DATA_BLOCK "1DB_simTT"   // DB999
{ S7_Optimized_Access := 'TRUE' }
VERSION : 0.1
   VAR
      TForSim : Array[0..359] of Int;   // Массив температур для эмуляции в формате Int
   END_VAR
BEGIN
   TForSim[0] := 200;
   TForSim[1] := 200;
   TForSim[2] := 199;
   TForSim[3] := 198;
   TForSim[4] := 197;
   TForSim[5] := 196;
   TForSim[6] := 196;
   TForSim[7] := 196;
   TForSim[8] := 196;
   TForSim[9] := 196;
   TForSim[10] := 195;
   TForSim[11] := 194;
   TForSim[12] := 194;
   TForSim[13] := 193;
   TForSim[14] := 193;
   TForSim[15] := 193;
   TForSim[16] := 193;
   TForSim[17] := 192;
   TForSim[18] := 192;
   TForSim[19] := 192;
   TForSim[20] := 192;
   TForSim[21] := 191;
   TForSim[22] := 191;
   TForSim[23] := 190;
   TForSim[24] := 189;
   TForSim[25] := 189;
   TForSim[26] := 189;
   TForSim[27] := 189;
   TForSim[28] := 188;
   TForSim[29] := 188;
   TForSim[30] := 187;
   TForSim[31] := 187;
   TForSim[32] := 187;
   TForSim[33] := 188;
   TForSim[34] := 188;
   TForSim[35] := 190;
   TForSim[36] := 190;
   TForSim[37] := 191;
   TForSim[38] := 191;
   TForSim[39] := 191;
   TForSim[40] := 193;
   TForSim[41] := 193;
   TForSim[42] := 193;
   TForSim[43] := 195;
   TForSim[44] := 195;
   TForSim[45] := 195;
   TForSim[46] := 196;
   TForSim[47] := 197;
   TForSim[48] := 198;
   TForSim[49] := 200;
   TForSim[50] := 200;
   TForSim[51] := 200;
   TForSim[52] := 201;
   TForSim[53] := 202;
   TForSim[54] := 203;
   TForSim[55] := 204;
   TForSim[56] := 205;
   TForSim[57] := 206;
   TForSim[58] := 207;
   TForSim[59] := 208;
   TForSim[60] := 209;
   TForSim[61] := 211;
   TForSim[62] := 211;
   TForSim[63] := 211;
   TForSim[64] := 211;
   TForSim[65] := 211;
   TForSim[66] := 210;
   TForSim[67] := 211;
   TForSim[68] := 211;
   TForSim[69] := 213;
   TForSim[70] := 214;
   TForSim[71] := 215;
   TForSim[72] := 215;
   TForSim[73] := 217;
   TForSim[74] := 218;
   TForSim[75] := 219;
   TForSim[76] := 220;
   TForSim[77] := 221;
   TForSim[78] := 222;
   TForSim[79] := 223;
   TForSim[80] := 225;
   TForSim[81] := 227;
   TForSim[82] := 230;
   TForSim[83] := 233;
   TForSim[84] := 236;
   TForSim[85] := 239;
   TForSim[86] := 241;
   TForSim[87] := 242;
   TForSim[88] := 244;
   TForSim[89] := 247;
   TForSim[90] := 249;
   TForSim[91] := 250;
   TForSim[92] := 250;
   TForSim[93] := 250;
   TForSim[94] := 250;
   TForSim[95] := 252;
   TForSim[96] := 254;
   TForSim[97] := 256;
   TForSim[98] := 257;
   TForSim[99] := 257;
   TForSim[100] := 259;
   TForSim[101] := 259;
   TForSim[102] := 259;
   TForSim[103] := 259;
   TForSim[104] := 260;
   TForSim[105] := 261;
   TForSim[106] := 261;
   TForSim[107] := 262;
   TForSim[108] := 262;
   TForSim[109] := 262;
   TForSim[110] := 263;
   TForSim[111] := 262;
   TForSim[112] := 262;
   TForSim[113] := 262;
   TForSim[114] := 262;
   TForSim[115] := 261;
   TForSim[116] := 261;
   TForSim[117] := 261;
   TForSim[118] := 261;
   TForSim[119] := 261;
   TForSim[120] := 260;
   TForSim[121] := 259;
   TForSim[122] := 259;
   TForSim[123] := 257;
   TForSim[124] := 256;
   TForSim[125] := 255;
   TForSim[126] := 254;
   TForSim[127] := 253;
   TForSim[128] := 253;
   TForSim[129] := 252;
   TForSim[130] := 252;
   TForSim[131] := 253;
   TForSim[132] := 253;
   TForSim[133] := 253;
   TForSim[134] := 252;
   TForSim[135] := 253;
   TForSim[136] := 253;
   TForSim[137] := 254;
   TForSim[138] := 255;
   TForSim[139] := 256;
   TForSim[140] := 259;
   TForSim[141] := 262;
   TForSim[142] := 264;
   TForSim[143] := 266;
   TForSim[144] := 266;
   TForSim[145] := 267;
   TForSim[146] := 267;
   TForSim[147] := 267;
   TForSim[148] := 270;
   TForSim[149] := 270;
   TForSim[150] := 271;
   TForSim[151] := 273;
   TForSim[152] := 273;
   TForSim[153] := 273;
   TForSim[154] := 274;
   TForSim[155] := 275;
   TForSim[156] := 275;
   TForSim[157] := 276;
   TForSim[158] := 277;
   TForSim[159] := 280;
   TForSim[160] := 281;
   TForSim[161] := 282;
   TForSim[162] := 282;
   TForSim[163] := 282;
   TForSim[164] := 284;
   TForSim[165] := 284;
   TForSim[166] := 285;
   TForSim[167] := 286;
   TForSim[168] := 286;
   TForSim[169] := 288;
   TForSim[170] := 288;
   TForSim[171] := 289;
   TForSim[172] := 291;
   TForSim[173] := 291;
   TForSim[174] := 292;
   TForSim[175] := 292;
   TForSim[176] := 292;
   TForSim[177] := 295;
   TForSim[178] := 294;
   TForSim[179] := 294;
   TForSim[180] := 295;
   TForSim[181] := 297;
   TForSim[182] := 298;
   TForSim[183] := 298;
   TForSim[184] := 300;
   TForSim[185] := 300;
   TForSim[186] := 300;
   TForSim[187] := 301;
   TForSim[188] := 301;
   TForSim[189] := 302;
   TForSim[190] := 303;
   TForSim[191] := 304;
   TForSim[192] := 304;
   TForSim[193] := 304;
   TForSim[194] := 306;
   TForSim[195] := 306;
   TForSim[196] := 306;
   TForSim[197] := 308;
   TForSim[198] := 307;
   TForSim[199] := 307;
   TForSim[200] := 309;
   TForSim[201] := 310;
   TForSim[202] := 311;
   TForSim[203] := 311;
   TForSim[204] := 312;
   TForSim[205] := 312;
   TForSim[206] := 312;
   TForSim[207] := 314;
   TForSim[208] := 313;
   TForSim[209] := 314;
   TForSim[210] := 314;
   TForSim[211] := 315;
   TForSim[212] := 315;
   TForSim[213] := 312;
   TForSim[214] := 312;
   TForSim[215] := 312;
   TForSim[216] := 312;
   TForSim[217] := 315;
   TForSim[218] := 315;
   TForSim[219] := 314;
   TForSim[220] := 313;
   TForSim[221] := 312;
   TForSim[222] := 311;
   TForSim[223] := 311;
   TForSim[224] := 311;
   TForSim[225] := 311;
   TForSim[226] := 311;
   TForSim[227] := 308;
   TForSim[228] := 309;
   TForSim[229] := 309;
   TForSim[230] := 308;
   TForSim[231] := 306;
   TForSim[232] := 305;
   TForSim[233] := 305;
   TForSim[234] := 303;
   TForSim[235] := 302;
   TForSim[236] := 302;
   TForSim[237] := 302;
   TForSim[238] := 301;
   TForSim[239] := 301;
   TForSim[240] := 301;
   TForSim[241] := 300;
   TForSim[242] := 299;
   TForSim[243] := 298;
   TForSim[244] := 297;
   TForSim[245] := 297;
   TForSim[246] := 297;
   TForSim[247] := 295;
   TForSim[248] := 295;
   TForSim[249] := 293;
   TForSim[250] := 293;
   TForSim[251] := 293;
   TForSim[252] := 290;
   TForSim[253] := 290;
   TForSim[254] := 289;
   TForSim[255] := 289;
   TForSim[256] := 289;
   TForSim[257] := 289;
   TForSim[258] := 290;
   TForSim[259] := 291;
   TForSim[260] := 292;
   TForSim[261] := 293;
   TForSim[262] := 294;
   TForSim[263] := 294;
   TForSim[264] := 295;
   TForSim[265] := 297;
   TForSim[266] := 298;
   TForSim[267] := 300;
   TForSim[268] := 301;
   TForSim[269] := 301;
   TForSim[270] := 302;
   TForSim[271] := 304;
   TForSim[272] := 304;
   TForSim[273] := 303;
   TForSim[274] := 301;
   TForSim[275] := 298;
   TForSim[276] := 299;
   TForSim[277] := 298;
   TForSim[278] := 296;
   TForSim[279] := 295;
   TForSim[280] := 295;
   TForSim[281] := 295;
   TForSim[282] := 294;
   TForSim[283] := 293;
   TForSim[284] := 292;
   TForSim[285] := 292;
   TForSim[286] := 290;
   TForSim[287] := 290;
   TForSim[288] := 287;
   TForSim[289] := 288;
   TForSim[290] := 288;
   TForSim[291] := 288;
   TForSim[292] := 286;
   TForSim[293] := 286;
   TForSim[294] := 284;
   TForSim[295] := 283;
   TForSim[296] := 280;
   TForSim[297] := 280;
   TForSim[298] := 278;
   TForSim[299] := 277;
   TForSim[300] := 276;
   TForSim[301] := 275;
   TForSim[302] := 274;
   TForSim[303] := 271;
   TForSim[304] := 272;
   TForSim[305] := 272;
   TForSim[306] := 270;
   TForSim[307] := 267;
   TForSim[308] := 265;
   TForSim[309] := 263;
   TForSim[310] := 261;
   TForSim[311] := 260;
   TForSim[312] := 258;
   TForSim[313] := 256;
   TForSim[314] := 254;
   TForSim[315] := 251;
   TForSim[316] := 252;
   TForSim[317] := 252;
   TForSim[318] := 253;
   TForSim[319] := 253;
   TForSim[320] := 251;
   TForSim[321] := 251;
   TForSim[322] := 249;
   TForSim[323] := 247;
   TForSim[324] := 246;
   TForSim[325] := 244;
   TForSim[326] := 242;
   TForSim[327] := 240;
   TForSim[328] := 238;
   TForSim[329] := 236;
   TForSim[330] := 233;
   TForSim[331] := 231;
   TForSim[332] := 229;
   TForSim[333] := 227;
   TForSim[334] := 225;
   TForSim[335] := 223;
   TForSim[336] := 222;
   TForSim[337] := 220;
   TForSim[338] := 219;
   TForSim[339] := 218;
   TForSim[340] := 217;
   TForSim[341] := 217;
   TForSim[342] := 217;
   TForSim[343] := 216;
   TForSim[344] := 215;
   TForSim[345] := 214;
   TForSim[346] := 214;
   TForSim[347] := 214;
   TForSim[348] := 213;
   TForSim[349] := 212;
   TForSim[350] := 210;
   TForSim[351] := 208;
   TForSim[352] := 206;
   TForSim[353] := 204;
   TForSim[354] := 203;
   TForSim[355] := 203;
   TForSim[356] := 203;
   TForSim[357] := 202;
   TForSim[358] := 202;
   TForSim[359] := 200;
END_DATA_BLOCK

// folder: System blocks/Program resources

DATA_BLOCK "Timer_2_DB"   // DB2
{ S7_Optimized_Access := 'TRUE' }
AUTHOR : Simatic
FAMILY : IEC
NAME : IEC_TMR
VERSION : 1.0
// stored: InstanceOfName IEC_TIMER
"IEC_TIMER"
BEGIN
END_DATA_BLOCK

DATA_BLOCK "IEC_Timer_1"   // DB601
{ S7_Optimized_Access := 'TRUE' }
AUTHOR : Simatic
FAMILY : IEC
NAME : IEC_TMR
VERSION : 1.0
// stored: InstanceOfName IEC_TIMER
"IEC_TIMER"
BEGIN
END_DATA_BLOCK

DATA_BLOCK "IEC_Timer_2"   // DB602
{ S7_Optimized_Access := 'TRUE' }
AUTHOR : Simatic
FAMILY : IEC
NAME : IEC_TMR
VERSION : 1.0
// stored: InstanceOfName IEC_TIMER
"IEC_TIMER"
BEGIN
END_DATA_BLOCK

DATA_BLOCK "IEC_Timer_3"   // DB603
{ S7_Optimized_Access := 'TRUE' }
AUTHOR : Simatic
FAMILY : IEC
NAME : IEC_TMR
VERSION : 1.0
// stored: InstanceOfName IEC_TIMER
"IEC_TIMER"
BEGIN
END_DATA_BLOCK

DATA_BLOCK "IEC_Timer_4"   // DB604
{ S7_Optimized_Access := 'TRUE' }
AUTHOR : Simatic
FAMILY : IEC
NAME : IEC_TMR
VERSION : 1.0
// stored: InstanceOfName IEC_TIMER
"IEC_TIMER"
BEGIN
END_DATA_BLOCK

DATA_BLOCK "IEC_Timer_5"   // DB605
{ S7_Optimized_Access := 'TRUE' }
AUTHOR : Simatic
FAMILY : IEC
NAME : IEC_TMR
VERSION : 1.0
// stored: InstanceOfName IEC_TIMER
"IEC_TIMER"
BEGIN
END_DATA_BLOCK

DATA_BLOCK "IEC_Timer_6"   // DB606
{ S7_Optimized_Access := 'TRUE' }
AUTHOR : Simatic
FAMILY : IEC
NAME : IEC_TMR
VERSION : 1.0
// stored: InstanceOfName IEC_TIMER
"IEC_TIMER"
BEGIN
END_DATA_BLOCK

DATA_BLOCK "IEC_Timer_7"   // DB607
{ S7_Optimized_Access := 'TRUE' }
AUTHOR : Simatic
FAMILY : IEC
NAME : IEC_TMR
VERSION : 1.0
// stored: InstanceOfName IEC_TIMER
"IEC_TIMER"
BEGIN
END_DATA_BLOCK

DATA_BLOCK "IEC_Timer_8"   // DB608
{ S7_Optimized_Access := 'TRUE' }
AUTHOR : Simatic
FAMILY : IEC
NAME : IEC_TMR
VERSION : 1.0
// stored: InstanceOfName IEC_TIMER
"IEC_TIMER"
BEGIN
END_DATA_BLOCK

DATA_BLOCK "SimTimer11"   // DB911
{ S7_Optimized_Access := 'TRUE' }
AUTHOR : Simatic
FAMILY : IEC
NAME : IEC_TMR
VERSION : 1.0
// stored: InstanceOfName IEC_TIMER
"IEC_TIMER"
BEGIN
END_DATA_BLOCK

DATA_BLOCK "SimTimer12"   // DB912
{ S7_Optimized_Access := 'TRUE' }
AUTHOR : Simatic
FAMILY : IEC
NAME : IEC_TMR
VERSION : 1.0
// stored: InstanceOfName IEC_TIMER
"IEC_TIMER"
BEGIN
END_DATA_BLOCK

DATA_BLOCK "SimTimer21"   // DB921
{ S7_Optimized_Access := 'TRUE' }
AUTHOR : Simatic
FAMILY : IEC
NAME : IEC_TMR
VERSION : 1.0
// stored: InstanceOfName IEC_TIMER
"IEC_TIMER"
BEGIN
END_DATA_BLOCK

DATA_BLOCK "SimTimer22"   // DB922
{ S7_Optimized_Access := 'TRUE' }
AUTHOR : Simatic
FAMILY : IEC
NAME : IEC_TMR
VERSION : 1.0
// stored: InstanceOfName IEC_TIMER
"IEC_TIMER"
BEGIN
END_DATA_BLOCK

// folder: (top level)

ORGANIZATION_BLOCK "1Main"   // OB1, LAD, ProgramCycle
TITLE = "Main Program Sweep (Cycle)"
{ S7_Optimized_Access := 'TRUE' }
VERSION : 0.1
// ОВ1 - главная циклическая программа. Вызывается операционной системой CPU
   VAR_INPUT
      Initial_Call : Bool;   // Initial call of this OB
      Remanence : Bool;   // =True, if remanent data are available
   END_VAR
   VAR_TEMP
      txExtStopVE : Bool;   // Внешняя блокировка дымососа по вибрации
      txExtStopTEB : Bool;   // Внешняя блокировка дымососа по т-ре подшипников
      txExtStopTEW : Bool;   // Внешняя блокировка дымососа по т-ре обмоток
      trValue : Real;   // Временная переменная типа Real
   END_VAR
BEGIN

REGION Network 2: Зеркалирование дискретных входов
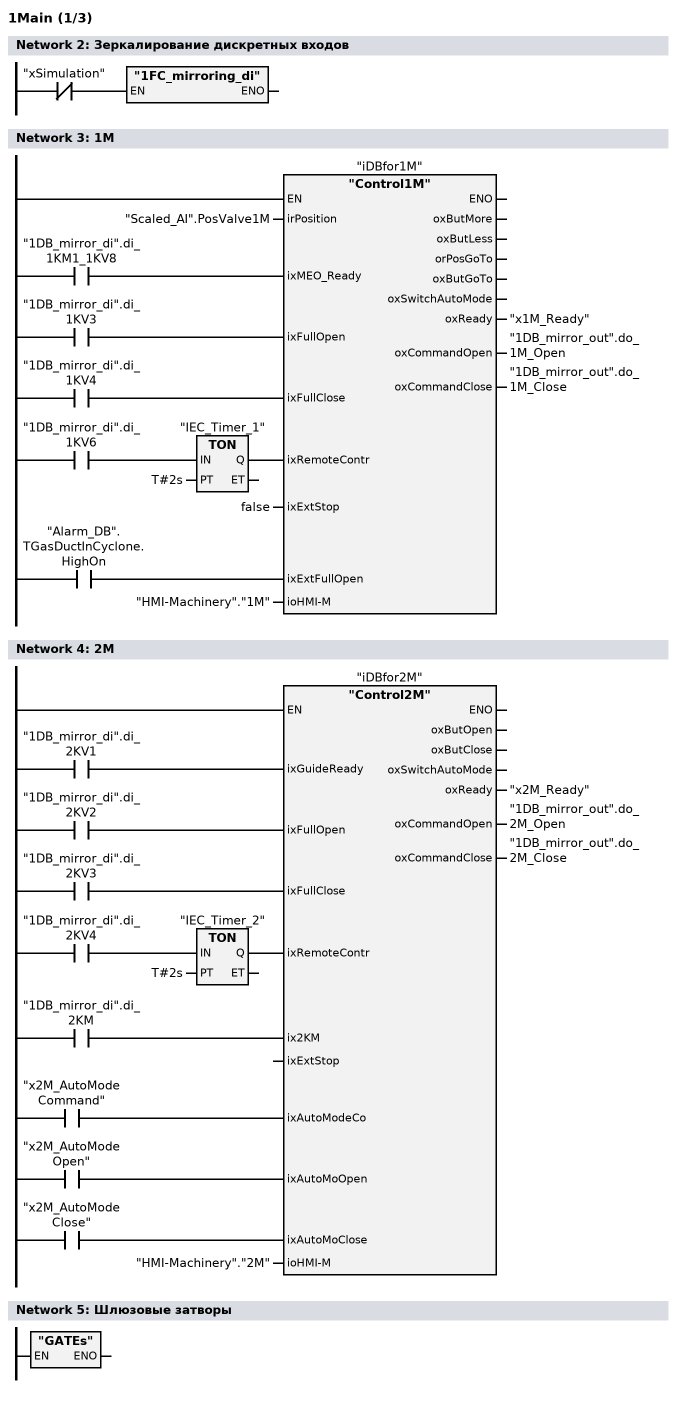
   RUNG wire#powerrail
      I_Contact( "xSimulation" )
      "1FC_mirroring_di"()
   END_RUNG
   // the same network as SCL:
   IF NOT "xSimulation" THEN "1FC_mirroring_di"(); END_IF;
END_REGION

REGION Network 3: 1M
   "IEC_Timer_1".TON(IN := "1DB_mirror_di".di_1KV6, PT := T#2s);
   "iDBfor1M"(irPosition := "Scaled_AI".PosValve1M,   // "Control1M"
              ixMEO_Ready := "1DB_mirror_di".di_1KM1_1KV8,
              ixFullOpen := "1DB_mirror_di".di_1KV3,
              ixFullClose := "1DB_mirror_di".di_1KV4,
              ixRemoteContr := "IEC_Timer_1".Q,
              ixExtStop := false,
              ixExtFullOpen := "Alarm_DB".TGasDuctInCyclone.HighOn,
              "ioHMI-M" := "HMI-Machinery"."1M",
              oxReady => "x1M_Ready",
              oxCommandOpen => "1DB_mirror_out".do_1M_Open,
              oxCommandClose => "1DB_mirror_out".do_1M_Close);
END_REGION

REGION Network 4: 2M
   "IEC_Timer_2".TON(IN := "1DB_mirror_di".di_2KV4, PT := T#2s);
   "iDBfor2M"(ixGuideReady := "1DB_mirror_di".di_2KV1,   // "Control2M"
              ixFullOpen := "1DB_mirror_di".di_2KV2,
              ixFullClose := "1DB_mirror_di".di_2KV3,
              ixRemoteContr := "IEC_Timer_2".Q,
              ix2KM := "1DB_mirror_di".di_2KM,
              ixAutoModeCo := "x2M_AutoModeCommand",
              ixAutoMoOpen := "x2M_AutoModeOpen",
              ixAutoMoClose := "x2M_AutoModeClose",
              "ioHMI-M" := "HMI-Machinery"."2M",
              oxReady => "x2M_Ready",
              oxCommandOpen => "1DB_mirror_out".do_2M_Open,
              oxCommandClose => "1DB_mirror_out".do_2M_Close);
END_REGION

REGION Network 5: Шлюзовые затворы
   RUNG wire#powerrail
      "GATEs"()
   END_RUNG
   // the same network as SCL:
   "GATEs"();
END_REGION

REGION Network 7: Подготовка внешних блокировок дымососа (14 шт.)
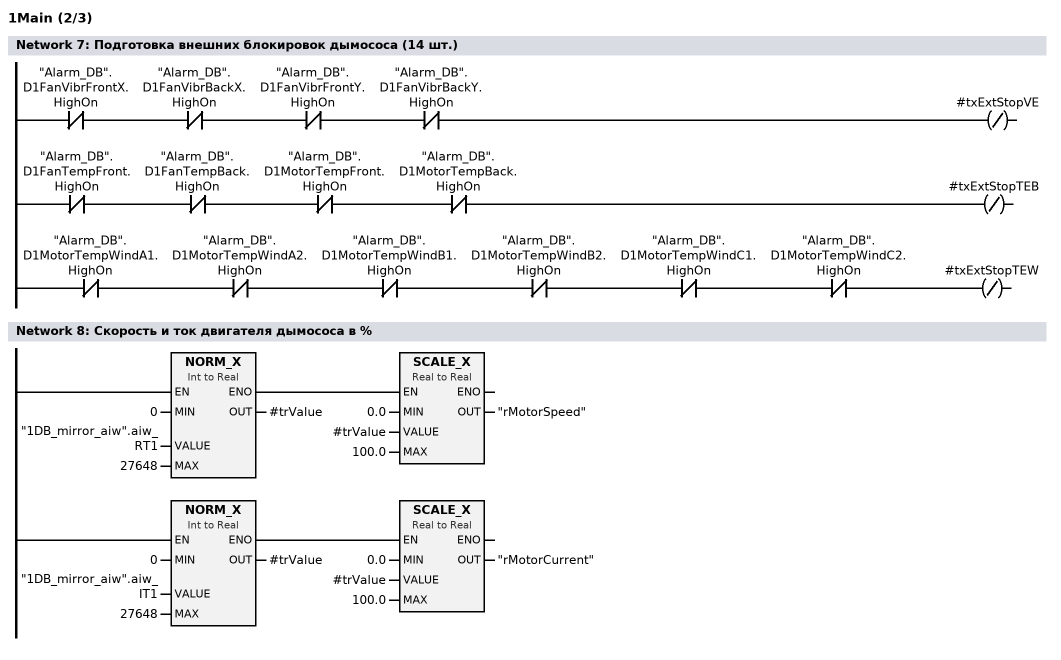
   RUNG wire#powerrail
      I_Contact( "Alarm_DB".D1FanVibrFrontX.HighOn )
      I_Contact( "Alarm_DB".D1FanVibrBackX.HighOn )
      I_Contact( "Alarm_DB".D1FanVibrFrontY.HighOn )
      I_Contact( "Alarm_DB".D1FanVibrBackY.HighOn )
      I_Coil( #txExtStopVE )
   END_RUNG
   RUNG wire#powerrail
      I_Contact( "Alarm_DB".D1FanTempFront.HighOn )
      I_Contact( "Alarm_DB".D1FanTempBack.HighOn )
      I_Contact( "Alarm_DB".D1MotorTempFront.HighOn )
      I_Contact( "Alarm_DB".D1MotorTempBack.HighOn )
      I_Coil( #txExtStopTEB )
   END_RUNG
   RUNG wire#powerrail
      I_Contact( "Alarm_DB".D1MotorTempWindA1.HighOn )
      I_Contact( "Alarm_DB".D1MotorTempWindA2.HighOn )
      I_Contact( "Alarm_DB".D1MotorTempWindB1.HighOn )
      I_Contact( "Alarm_DB".D1MotorTempWindB2.HighOn )
      I_Contact( "Alarm_DB".D1MotorTempWindC1.HighOn )
      I_Contact( "Alarm_DB".D1MotorTempWindC2.HighOn )
      I_Coil( #txExtStopTEW )
   END_RUNG
   // the same network as SCL:
   #txExtStopVE := NOT (NOT "Alarm_DB".D1FanVibrFrontX.HighOn AND NOT "Alarm_DB".D1FanVibrBackX.HighOn AND NOT "Alarm_DB".D1FanVibrFrontY.HighOn AND NOT "Alarm_DB".D1FanVibrBackY.HighOn);
   #txExtStopTEB := NOT (NOT "Alarm_DB".D1FanTempFront.HighOn AND NOT "Alarm_DB".D1FanTempBack.HighOn AND NOT "Alarm_DB".D1MotorTempFront.HighOn AND NOT "Alarm_DB".D1MotorTempBack.HighOn);
   #txExtStopTEW := NOT (NOT "Alarm_DB".D1MotorTempWindA1.HighOn AND NOT "Alarm_DB".D1MotorTempWindA2.HighOn AND NOT "Alarm_DB".D1MotorTempWindB1.HighOn AND NOT "Alarm_DB".D1MotorTempWindB2.HighOn AND NOT "Alarm_DB".D1MotorTempWindC1.HighOn AND NOT "Alarm_DB".D1MotorTempWindC2.HighOn);
END_REGION

REGION Network 8: Скорость и ток двигателя дымососа в %
   RUNG wire#powerrail
      { S7_Templates := "[SrcType := Int, DestType := Real]" } Normalize(min := 0, value := "1DB_mirror_aiw".aiw_RT1, max := 27648, out => #trValue)
      { S7_Templates := "[SrcType := Real, DestType := Real]" } Scale(min := 0.0, value := #trValue, max := 100.0, out => "rMotorSpeed")
   END_RUNG
   RUNG wire#powerrail
      { S7_Templates := "[SrcType := Int, DestType := Real]" } Normalize(min := 0, value := "1DB_mirror_aiw".aiw_IT1, max := 27648, out => #trValue)
      { S7_Templates := "[SrcType := Real, DestType := Real]" } Scale(min := 0.0, value := #trValue, max := 100.0, out => "rMotorCurrent")
   END_RUNG
   // the same network as SCL:
   #trValue := NORM_X(MIN := 0, VALUE := "1DB_mirror_aiw".aiw_RT1, MAX := 27648);
   "rMotorSpeed" := SCALE_X(MIN := 0.0, VALUE := #trValue, MAX := 100.0);
   #trValue := NORM_X(MIN := 0, VALUE := "1DB_mirror_aiw".aiw_IT1, MAX := 27648);
   "rMotorCurrent" := SCALE_X(MIN := 0.0, VALUE := #trValue, MAX := 100.0);
END_REGION

REGION Network 9: Дымосос
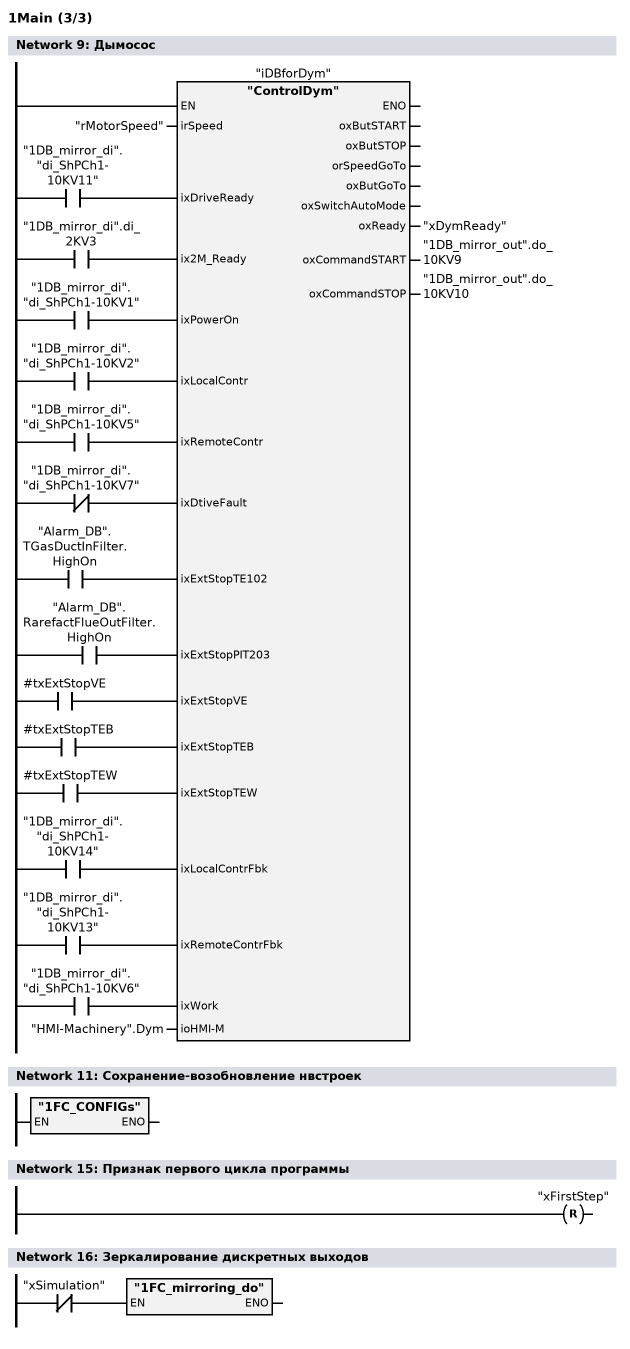
   RUNG wire#powerrail
      "iDBforDym"(ixDriveReady := wire#w1, ix2M_Ready := wire#w2, ixPowerOn := wire#w3, ixLocalContr := wire#w4, ixRemoteContr := wire#w5, ixDtiveFault := wire#w6, ixExtStopTE102 := wire#w7, ixExtStopРІТ203 := wire#w8, ixExtStopVE := wire#w9, ixExtStopTEB := wire#w10, ixExtStopTEW := wire#w11, ixLocalContrFbk := wire#w12, ixRemoteContrFbk := wire#w13, ixWork := wire#w14, irSpeed := "rMotorSpeed", "ioHMI-M" := "HMI-Machinery".Dym, oxButSTART =>, oxButSTOP =>, orSpeedGoTo =>, oxButGoTo =>, oxSwitchAutoMode =>, oxReady => "xDymReady", oxCommandSTART => "1DB_mirror_out".do_10KV9, oxCommandSTOP => "1DB_mirror_out".do_10KV10)
   END_RUNG
   RUNG wire#powerrail
      Contact( "1DB_mirror_di"."di_ShPCh1-10KV11" )
   END_RUNG wire#w1
   RUNG wire#powerrail
      Contact( "1DB_mirror_di".di_2KV3 )
   END_RUNG wire#w2
   RUNG wire#powerrail
      Contact( "1DB_mirror_di"."di_ShPCh1-10KV1" )
   END_RUNG wire#w3
   RUNG wire#powerrail
      Contact( "1DB_mirror_di"."di_ShPCh1-10KV2" )
   END_RUNG wire#w4
   RUNG wire#powerrail
      Contact( "1DB_mirror_di"."di_ShPCh1-10KV5" )
   END_RUNG wire#w5
   RUNG wire#powerrail
      I_Contact( "1DB_mirror_di"."di_ShPCh1-10KV7" )
   END_RUNG wire#w6
   RUNG wire#powerrail
      Contact( "Alarm_DB".TGasDuctInFilter.HighOn )
   END_RUNG wire#w7
   RUNG wire#powerrail
      Contact( "Alarm_DB".RarefactFlueOutFilter.HighOn )
   END_RUNG wire#w8
   RUNG wire#powerrail
      Contact( #txExtStopVE )
   END_RUNG wire#w9
   RUNG wire#powerrail
      Contact( #txExtStopTEB )
   END_RUNG wire#w10
   RUNG wire#powerrail
      Contact( #txExtStopTEW )
   END_RUNG wire#w11
   RUNG wire#powerrail
      Contact( "1DB_mirror_di"."di_ShPCh1-10KV14" )
   END_RUNG wire#w12
   RUNG wire#powerrail
      Contact( "1DB_mirror_di"."di_ShPCh1-10KV13" )
   END_RUNG wire#w13
   RUNG wire#powerrail
      Contact( "1DB_mirror_di"."di_ShPCh1-10KV6" )
   END_RUNG wire#w14
   // the same network as SCL:
   "iDBforDym"(irSpeed := "rMotorSpeed",   // "ControlDym"
               ixDriveReady := "1DB_mirror_di"."di_ShPCh1-10KV11",
               ix2M_Ready := "1DB_mirror_di".di_2KV3,
               ixPowerOn := "1DB_mirror_di"."di_ShPCh1-10KV1",
               ixLocalContr := "1DB_mirror_di"."di_ShPCh1-10KV2",
               ixRemoteContr := "1DB_mirror_di"."di_ShPCh1-10KV5",
               ixDtiveFault := NOT "1DB_mirror_di"."di_ShPCh1-10KV7",
               ixExtStopTE102 := "Alarm_DB".TGasDuctInFilter.HighOn,
               ixExtStopРІТ203 := "Alarm_DB".RarefactFlueOutFilter.HighOn,
               ixExtStopVE := #txExtStopVE,
               ixExtStopTEB := #txExtStopTEB,
               ixExtStopTEW := #txExtStopTEW,
               ixLocalContrFbk := "1DB_mirror_di"."di_ShPCh1-10KV14",
               ixRemoteContrFbk := "1DB_mirror_di"."di_ShPCh1-10KV13",
               ixWork := "1DB_mirror_di"."di_ShPCh1-10KV6",
               "ioHMI-M" := "HMI-Machinery".Dym,
               oxReady => "xDymReady",
               oxCommandSTART => "1DB_mirror_out".do_10KV9,
               oxCommandSTOP => "1DB_mirror_out".do_10KV10);
END_REGION

REGION Network 11: Сохранение-возобновление нвстроек
   RUNG wire#powerrail
      "1FC_CONFIGs"()
   END_RUNG
   // the same network as SCL:
   "1FC_CONFIGs"();
END_REGION

REGION Network 14: Все NW что ниже должны быть в конце ОВ1:
END_REGION

REGION Network 15: Признак первого цикла программы
   RUNG wire#powerrail
      R_Coil( "xFirstStep" )
   END_RUNG
   // the same network as SCL:
   "xFirstStep" := FALSE;
END_REGION

REGION Network 16: Зеркалирование дискретных выходов
   RUNG wire#powerrail
      I_Contact( "xSimulation" )
      "1FC_mirroring_do"()
   END_RUNG
   // the same network as SCL:
   IF NOT "xSimulation" THEN "1FC_mirroring_do"(); END_IF;
END_REGION
END_ORGANIZATION_BLOCK

ORGANIZATION_BLOCK "1Cyclic irupt_100"   // OB30, LAD, CyclicInterrupt
TITLE = "Cyclic interrupt"
{ S7_Optimized_Access := 'TRUE' }
VERSION : 0.1
// ОВ30 настроен на циклический вызов каждые 100 милисекунд. 
// Вызывается операционной системой CPU
   VAR_INPUT
      Initial_Call : Bool;   // Initial call of this OB
      Event_Count : Int;   // Events discarded
   END_VAR
   VAR_TEMP
      trForRegeneration : Real;   // Разность разрежений
      tiDymPID_Command : Int;   // Для задания скорости приводу дымососа от ПИДа
   END_VAR
   VAR_TEMP   // added for the SCL form of the ladder/FBD networks
      _w1 : Bool;
      _w2 : Bool;
      _w3 : Bool;
      _w4 : Bool;
   END_VAR
BEGIN

REGION Network 2: Симуляция механизмов
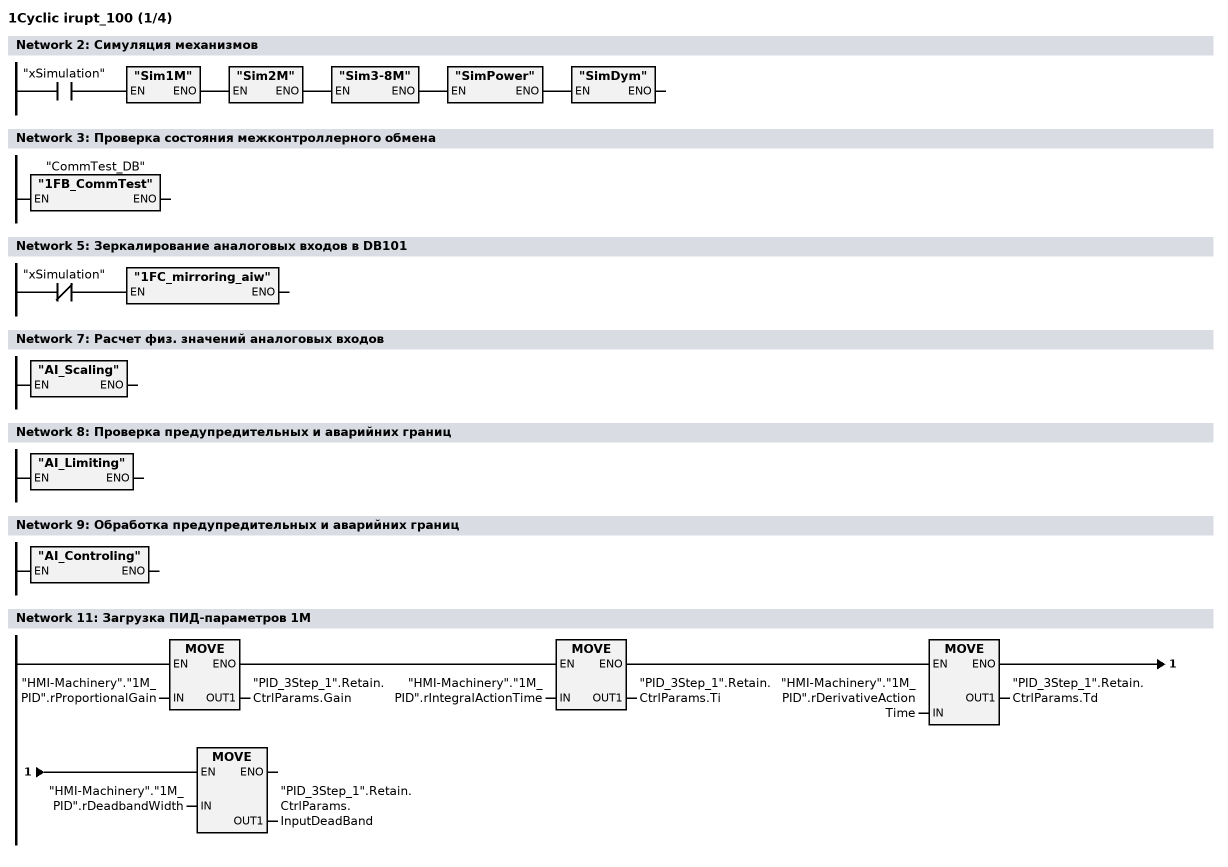
   RUNG wire#powerrail
      Contact( "xSimulation" )
      "Sim1M"()
      "Sim2M"()
      "Sim3-8M"()
      "SimPower"()
      "SimDym"()
   END_RUNG
   // the same network as SCL:
   "Sim1M"(EN := "xSimulation", ENO => #_w1);
   "Sim2M"(EN := #_w1, ENO => #_w2);
   "Sim3-8M"(EN := #_w2, ENO => #_w3);
   "SimPower"(EN := #_w3, ENO => #_w4);
   IF #_w4 THEN "SimDym"(); END_IF;
END_REGION

REGION Network 3: Проверка состояния межконтроллерного обмена
   RUNG wire#powerrail
      "CommTest_DB"()
   END_RUNG
   // the same network as SCL:
   "CommTest_DB"();   // "1FB_CommTest"
END_REGION

REGION Network 5: Зеркалирование аналоговых входов в DB101
   RUNG wire#powerrail
      I_Contact( "xSimulation" )
      "1FC_mirroring_aiw"()
   END_RUNG
   // the same network as SCL:
   IF NOT "xSimulation" THEN "1FC_mirroring_aiw"(); END_IF;
END_REGION

REGION Network 6: Обработка аналоговых входов (networks 4-6)
END_REGION

REGION Network 7: Расчет физ. значений аналоговых входов
   RUNG wire#powerrail
      "AI_Scaling"()
   END_RUNG
   // the same network as SCL:
   "AI_Scaling"();
END_REGION

REGION Network 8: Проверка предупредительных и аварийних границ
   RUNG wire#powerrail
      "AI_Limiting"()
   END_RUNG
   // the same network as SCL:
   "AI_Limiting"();
END_REGION

REGION Network 9: Обработка предупредительных и аварийних границ
   RUNG wire#powerrail
      "AI_Controling"()
   END_RUNG
   // the same network as SCL:
   "AI_Controling"();
END_REGION

REGION Network 11: Загрузка ПИД-параметров 1M
   RUNG wire#powerrail
      Move(in := "HMI-Machinery"."1M_PID".rProportionalGain, out1 => "PID_3Step_1".Retain.CtrlParams.Gain)
      Move(in := "HMI-Machinery"."1M_PID".rIntegralActionTime, out1 => "PID_3Step_1".Retain.CtrlParams.Ti)
      Move(in := "HMI-Machinery"."1M_PID".rDerivativeActionTime, out1 => "PID_3Step_1".Retain.CtrlParams.Td)
      Move(in := "HMI-Machinery"."1M_PID".rDeadbandWidth, out1 => "PID_3Step_1".Retain.CtrlParams.InputDeadBand)
   END_RUNG
   // the same network as SCL:
   "PID_3Step_1".Retain.CtrlParams.Gain := "HMI-Machinery"."1M_PID".rProportionalGain;
   "PID_3Step_1".Retain.CtrlParams.Ti := "HMI-Machinery"."1M_PID".rIntegralActionTime;
   "PID_3Step_1".Retain.CtrlParams.Td := "HMI-Machinery"."1M_PID".rDerivativeActionTime;
   "PID_3Step_1".Retain.CtrlParams.InputDeadBand := "HMI-Machinery"."1M_PID".rDeadbandWidth;
END_REGION

REGION Network 12: ПИД-регурятор для 1М
   // Жоден з цих трьох ПІДів (що нижче) не працюють у PLCSIM. Одже остаточне налагодження можливе тільке на майданчику
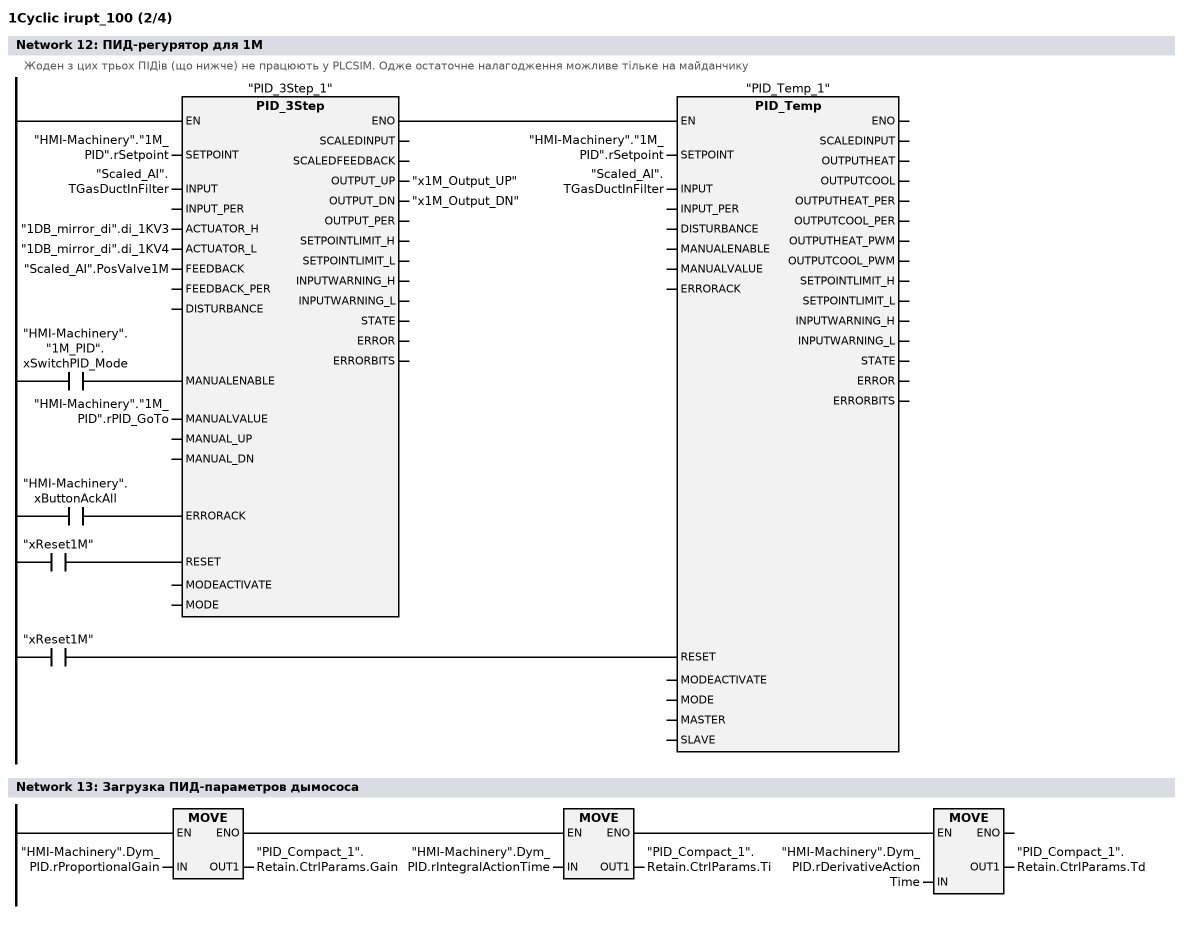
   // ENO of a box is taken as its EN; it also drops when the box reports an error
   "PID_3Step_1"(Setpoint := "HMI-Machinery"."1M_PID".rSetpoint,   // PID_3Step
                 Input := "Scaled_AI".TGasDuctInFilter,
                 Actuator_H := "1DB_mirror_di".di_1KV3,
                 Actuator_L := "1DB_mirror_di".di_1KV4,
                 Feedback := "Scaled_AI".PosValve1M,
                 ManualEnable := "HMI-Machinery"."1M_PID".xSwitchPID_Mode,
                 ManualValue := "HMI-Machinery"."1M_PID".rPID_GoTo,
                 ErrorAck := "HMI-Machinery".xButtonAckAll,
                 Reset := "xReset1M",
                 Output_UP => "x1M_Output_UP",
                 Output_DN => "x1M_Output_DN");
   "PID_Temp_1"(Setpoint := "HMI-Machinery"."1M_PID".rSetpoint,   // PID_Temp
                Input := "Scaled_AI".TGasDuctInFilter,
                Reset := "xReset1M");
END_REGION

REGION Network 13: Загрузка ПИД-параметров дымососа
   RUNG wire#powerrail
      Move(in := "HMI-Machinery".Dym_PID.rProportionalGain, out1 => "PID_Compact_1".Retain.CtrlParams.Gain)
      Move(in := "HMI-Machinery".Dym_PID.rIntegralActionTime, out1 => "PID_Compact_1".Retain.CtrlParams.Ti)
      Move(in := "HMI-Machinery".Dym_PID.rDerivativeActionTime, out1 => "PID_Compact_1".Retain.CtrlParams.Td)
   END_RUNG
   // the same network as SCL:
   "PID_Compact_1".Retain.CtrlParams.Gain := "HMI-Machinery".Dym_PID.rProportionalGain;
   "PID_Compact_1".Retain.CtrlParams.Ti := "HMI-Machinery".Dym_PID.rIntegralActionTime;
   "PID_Compact_1".Retain.CtrlParams.Td := "HMI-Machinery".Dym_PID.rDerivativeActionTime;
END_REGION

REGION Network 14: ПИД-регурятор для дымососа
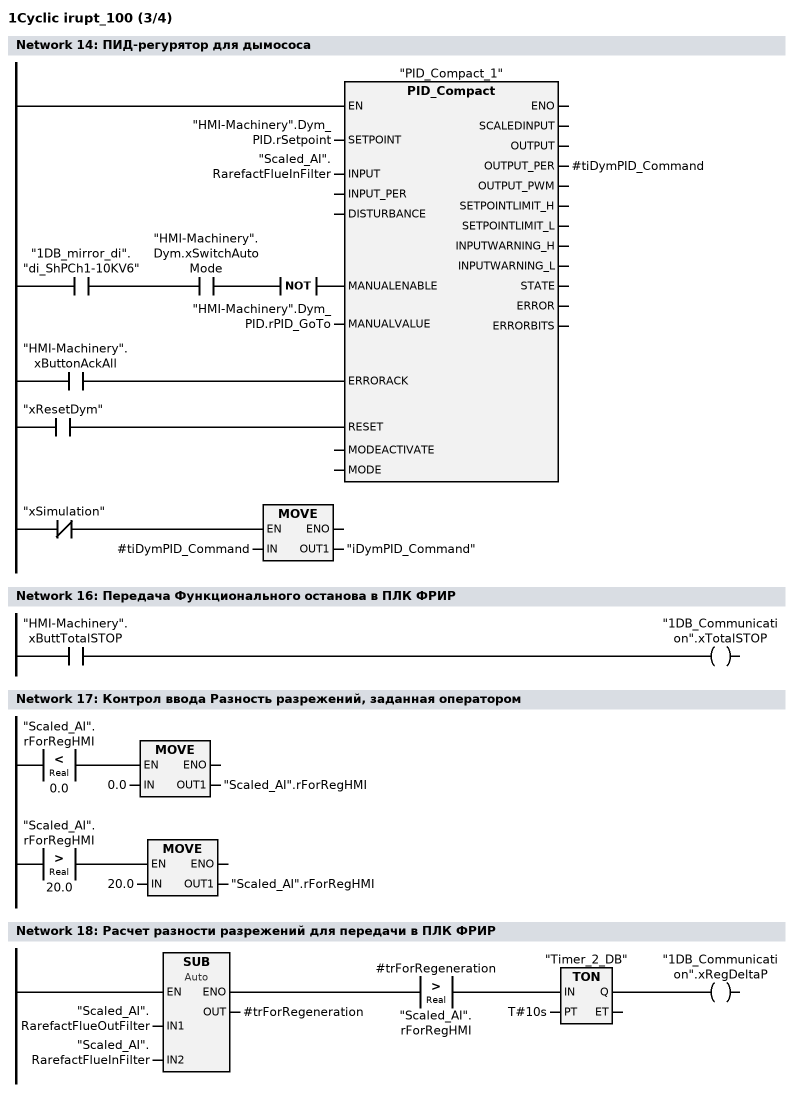
   "PID_Compact_1"(Setpoint := "HMI-Machinery".Dym_PID.rSetpoint,   // PID_Compact
                   Input := "Scaled_AI".RarefactFlueInFilter,
                   ManualEnable := NOT ("1DB_mirror_di"."di_ShPCh1-10KV6" AND "HMI-Machinery".Dym.xSwitchAutoMode),
                   ManualValue := "HMI-Machinery".Dym_PID.rPID_GoTo,
                   ErrorAck := "HMI-Machinery".xButtonAckAll,
                   Reset := "xResetDym",
                   Output_PER => #tiDymPID_Command);
   IF NOT "xSimulation" THEN "iDymPID_Command" := #tiDymPID_Command; END_IF;
END_REGION

REGION Network 16: Передача Функционального останова в ПЛК ФРИР
   RUNG wire#powerrail
      Contact( "HMI-Machinery".xButtTotalSTOP )
      Coil( "1DB_Communication".xTotalSTOP )
   END_RUNG
   // the same network as SCL:
   "1DB_Communication".xTotalSTOP := "HMI-Machinery".xButtTotalSTOP;
END_REGION

REGION Network 17: Контрол ввода Разность разрежений, заданная оператором
   RUNG wire#powerrail
      { S7_Templates := "SrcType := Real" } LT_Contact(in1 := "Scaled_AI".rForRegHMI, in2 := 0.0)
      Move(in := 0.0, out1 => "Scaled_AI".rForRegHMI)
   END_RUNG
   RUNG wire#powerrail
      { S7_Templates := "SrcType := Real" } GT_Contact(in1 := "Scaled_AI".rForRegHMI, in2 := 20.0)
      Move(in := 20.0, out1 => "Scaled_AI".rForRegHMI)
   END_RUNG
   // the same network as SCL:
   IF "Scaled_AI".rForRegHMI < 0.0 THEN "Scaled_AI".rForRegHMI := 0.0; END_IF;
   IF "Scaled_AI".rForRegHMI > 20.0 THEN "Scaled_AI".rForRegHMI := 20.0; END_IF;
END_REGION

REGION Network 18: Расчет разности разрежений для передачи в ПЛК ФРИР
   #trForRegeneration := "Scaled_AI".RarefactFlueOutFilter - "Scaled_AI".RarefactFlueInFilter;
   "Timer_2_DB".TON(IN := #trForRegeneration > "Scaled_AI".rForRegHMI, PT := T#10s);
   "1DB_Communication".xRegDeltaP := "Timer_2_DB".Q;
END_REGION

REGION Network 19: Передача данных в контроллер ФРИР
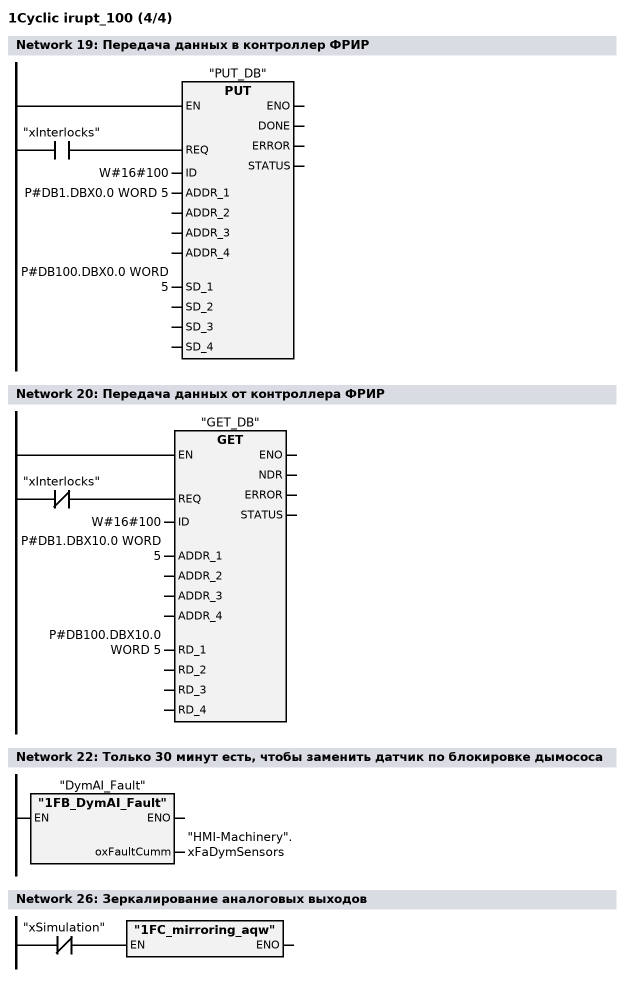
   "PUT_DB"(REQ := "xInterlocks", ID := W#16#100, ADDR_1 := P#DB1.DBX0.0 WORD 5, SD_1 := P#DB100.DBX0.0 WORD 5);   // PUT
END_REGION

REGION Network 20: Передача данных от контроллера ФРИР
   "GET_DB"(REQ := NOT "xInterlocks",   // GET
            ID := W#16#100,
            ADDR_1 := P#DB1.DBX10.0 WORD 5,
            RD_1 := P#DB100.DBX10.0 WORD 5);
END_REGION

REGION Network 22: Только 30 минут есть, чтобы заменить датчик по блокировке дымососа
   RUNG wire#powerrail
      "DymAI_Fault"(oxFaultCumm => "HMI-Machinery".xFaDymSensors)
   END_RUNG
   // the same network as SCL:
   "DymAI_Fault"(oxFaultCumm => "HMI-Machinery".xFaDymSensors);   // "1FB_DymAI_Fault"
END_REGION

REGION Network 25: Все NW что ниже должны быть в конце ОВ30:
END_REGION

REGION Network 26: Зеркалирование аналоговых выходов
   RUNG wire#powerrail
      I_Contact( "xSimulation" )
      "1FC_mirroring_aqw"()
   END_RUNG
   // the same network as SCL:
   IF NOT "xSimulation" THEN "1FC_mirroring_aqw"(); END_IF;
END_REGION
END_ORGANIZATION_BLOCK

ORGANIZATION_BLOCK "1Cyclic irupt_1000"   // OB31, LAD, CyclicInterrupt
TITLE = "Cyclic interrupt"
{ S7_Optimized_Access := 'TRUE' }
VERSION : 0.1
// ОВ31 настроен на циклический вызов каждые 1000 милисекунд. Вызывается операционной системой CPU
   VAR_INPUT
      Initial_Call : Bool;   // Initial call of this OB
      Event_Count : Int;   // Events discarded
   END_VAR
   VAR_TEMP
      tdtL : DTL;
      tiRetVal : Int;
      ttim : Time;
      tdi : DInt;
   END_VAR
BEGIN

REGION Network 2: Симуляция для A1.02... A1.06
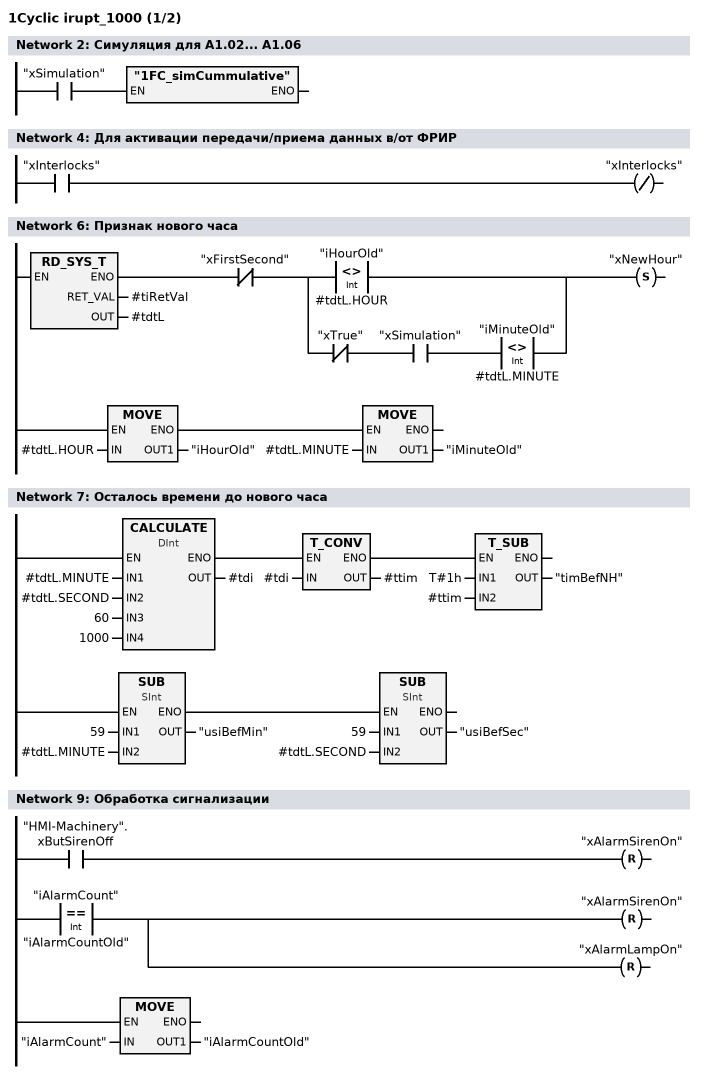
   RUNG wire#powerrail
      Contact( "xSimulation" )
      "1FC_simCummulative"()
   END_RUNG
   // the same network as SCL:
   IF "xSimulation" THEN "1FC_simCummulative"(); END_IF;
END_REGION

REGION Network 4: Для активации передачи/приема данных в/от ФРИР
   RUNG wire#powerrail
      Contact( "xInterlocks" )
      I_Coil( "xInterlocks" )
   END_RUNG
   // the same network as SCL:
   "xInterlocks" := NOT "xInterlocks";
END_REGION

REGION Network 6: Признак нового часа
   // ENO of a box is taken as its EN; it also drops when the box reports an error
   #tiRetVal := RD_SYS_T(OUT => #tdtL);
   IF NOT "xFirstSecond" AND (("iHourOld" <> #tdtL.HOUR) OR (NOT "xTrue" AND "xSimulation" AND ("iMinuteOld" <> #tdtL.MINUTE))) THEN
       "xNewHour" := TRUE;
   END_IF;
   "iHourOld" := #tdtL.HOUR;
   "iMinuteOld" := #tdtL.MINUTE;
END_REGION

REGION Network 7: Осталось времени до нового часа
   // ENO of a box is taken as its EN; it also drops when the box reports an error
   #tdi := (#tdtL.MINUTE*60+#tdtL.SECOND)*1000;
   #ttim := T_CONV(IN := #tdi);
   "timBefNH" := T_SUB(IN1 := T#1h, IN2 := #ttim);
   "usiBefMin" := 59 - #tdtL.MINUTE;
   "usiBefSec" := 59 - #tdtL.SECOND;
END_REGION

REGION Network 9: Обработка сигнализации
   RUNG wire#powerrail
      Contact( "HMI-Machinery".xButSirenOff )
      R_Coil( "xAlarmSirenOn" )
   END_RUNG
   RUNG wire#powerrail
      { S7_Templates := "SrcType := Int" } EQ_Contact(in1 := "iAlarmCount", in2 := "iAlarmCountOld")
      wire#w1
      R_Coil( "xAlarmSirenOn" )
   END_RUNG
   RUNG wire#w1
      R_Coil( "xAlarmLampOn" )
   END_RUNG
   RUNG wire#powerrail
      Move(in := "iAlarmCount", out1 => "iAlarmCountOld")
   END_RUNG
   // the same network as SCL:
   IF "HMI-Machinery".xButSirenOff THEN "xAlarmSirenOn" := FALSE; END_IF;
   IF "iAlarmCount" = "iAlarmCountOld" THEN
       "xAlarmSirenOn" := FALSE;
       "xAlarmLampOn" := FALSE;
   END_IF;
   "iAlarmCountOld" := "iAlarmCount";
END_REGION

REGION Network 10: Мигающий характер световой сигнализации
   // Немигающий звук
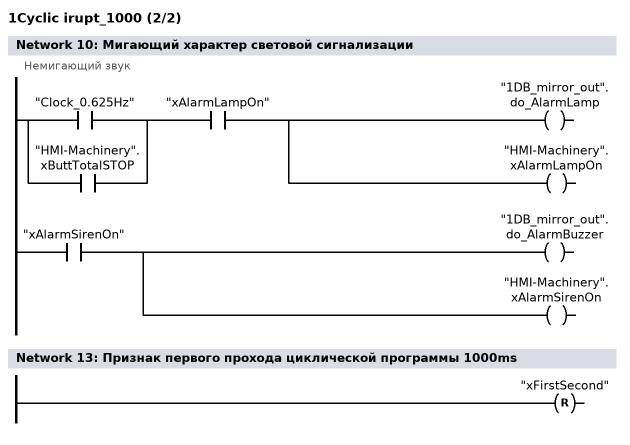
   RUNG wire#powerrail
      Contact( "Clock_0.625Hz" )
      wire#w1
      Contact( "xAlarmLampOn" )
      wire#w2
      Coil( "1DB_mirror_out".do_AlarmLamp )
   END_RUNG
   RUNG wire#powerrail
      Contact( "HMI-Machinery".xButtTotalSTOP )
   END_RUNG wire#w1
   RUNG wire#w2
      Coil( "HMI-Machinery".xAlarmLampOn )
   END_RUNG
   RUNG wire#powerrail
      Contact( "xAlarmSirenOn" )
      wire#w3
      Coil( "1DB_mirror_out".do_AlarmBuzzer )
   END_RUNG
   RUNG wire#w3
      Coil( "HMI-Machinery".xAlarmSirenOn )
   END_RUNG
   // the same network as SCL:
   "1DB_mirror_out".do_AlarmLamp := ("Clock_0.625Hz" OR "HMI-Machinery".xButtTotalSTOP) AND "xAlarmLampOn";
   "HMI-Machinery".xAlarmLampOn := "1DB_mirror_out".do_AlarmLamp;
   "1DB_mirror_out".do_AlarmBuzzer := "xAlarmSirenOn";
   "HMI-Machinery".xAlarmSirenOn := "xAlarmSirenOn";
END_REGION

REGION Network 12: Все NW что ниже должны быть в конце ОВ31:
END_REGION

REGION Network 13: Признак первого прохода циклической программы 1000ms
   RUNG wire#powerrail
      R_Coil( "xFirstSecond" )
   END_RUNG
   // the same network as SCL:
   "xFirstSecond" := FALSE;
END_REGION
END_ORGANIZATION_BLOCK

ORGANIZATION_BLOCK "1Cyclic interrupt_3000"   // OB33, LAD, CyclicInterrupt
{ S7_Optimized_Access := 'TRUE' }
VERSION : 0.1
   VAR_INPUT
      Initial_Call : Bool;   // Initial call of this OB
      Event_Count : Int;   // Events discarded
   END_VAR
BEGIN

REGION Network 2: Прошло три секунды
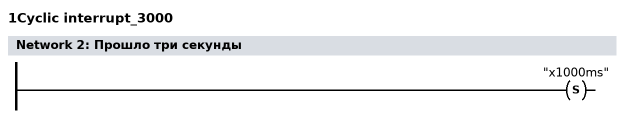
   RUNG wire#powerrail
      S_Coil( "x1000ms" )
   END_RUNG
   // the same network as SCL:
   "x1000ms" := TRUE;
END_REGION
END_ORGANIZATION_BLOCK

ORGANIZATION_BLOCK "1Startup"   // OB100, LAD, Startup
TITLE = "Complete Restart"
{ S7_Optimized_Access := 'TRUE' }
VERSION : 0.1
// ОВ100 -  вызывается однократно операционной системой CPU при старте CPU
   VAR_INPUT
      LostRetentive : Bool;   // True if retentive data are lost
      LostRTC : Bool;   // True if date and time are lost
   END_VAR
BEGIN

REGION Network 2: Логическая единица
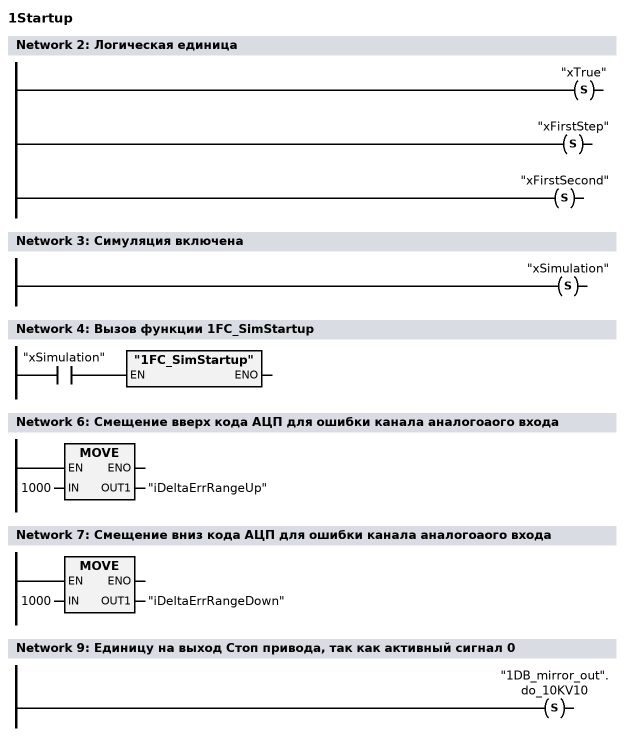
   RUNG wire#powerrail
      S_Coil( "xTrue" )
   END_RUNG
   RUNG wire#powerrail
      S_Coil( "xFirstStep" )
   END_RUNG
   RUNG wire#powerrail
      S_Coil( "xFirstSecond" )
   END_RUNG
   // the same network as SCL:
   "xTrue" := TRUE;
   "xFirstStep" := TRUE;
   "xFirstSecond" := TRUE;
END_REGION

REGION Network 3: Симуляция включена
   RUNG wire#powerrail
      S_Coil( "xSimulation" )
   END_RUNG
   // the same network as SCL:
   "xSimulation" := TRUE;
END_REGION

REGION Network 4: Вызов функции 1FC_SimStartup
   RUNG wire#powerrail
      Contact( "xSimulation" )
      "1FC_SimStartup"()
   END_RUNG
   // the same network as SCL:
   IF "xSimulation" THEN "1FC_SimStartup"(); END_IF;
END_REGION

REGION Network 6: Смещение вверх кода АЦП для ошибки канала аналогоаого входа
   RUNG wire#powerrail
      Move(in := 1000, out1 => "iDeltaErrRangeUp")
   END_RUNG
   // the same network as SCL:
   "iDeltaErrRangeUp" := 1000;
END_REGION

REGION Network 7: Смещение вниз кода АЦП для ошибки канала аналогоаого входа
   RUNG wire#powerrail
      Move(in := 1000, out1 => "iDeltaErrRangeDown")
   END_RUNG
   // the same network as SCL:
   "iDeltaErrRangeDown" := 1000;
END_REGION

REGION Network 9: Единицу на выход Стоп привода, так как активный сигнал 0
   RUNG wire#powerrail
      S_Coil( "1DB_mirror_out".do_10KV10 )
   END_RUNG
   // the same network as SCL:
   "1DB_mirror_out".do_10KV10 := TRUE;
END_REGION
END_ORGANIZATION_BLOCK

// folder: ERRORs

FUNCTION_BLOCK "1FB_DymAI_Fault"   // FB99, LAD
{ S7_Optimized_Access := 'TRUE' }
VERSION : 0.1
   VAR_OUTPUT
      oxFaultCumm : Bool;
   END_VAR
   VAR
      siTotalFault : Int;   // Всего аварий
      sxArrayP : Array[0..48] of Bool;   // Обнаружение Фронта
      sxN1 : Bool;   // Обнаружение Фронта
      sxFaultCumm : Bool;   // Сборная авария
      IEC_Timer_0_Instance : TON_TIME;
   END_VAR
   VAR_TEMP
      txNoFault : Bool;   // Группировка отсутствия аварии
      ttimBC : Time;   // Обратный отсчет в формате Time
      tdiBC : DInt;   // Сконвертированное время
      tdiTT : DInt;   // Временная переменная
      ttimHalfHour : Time;   // Для симуляции
   END_VAR
   VAR CONSTANT
      ctimHalfHour : Time := T#30M;   // 30 минут
   END_VAR
   VAR_TEMP   // added for the SCL form of the ladder/FBD networks
      _w1 : Bool;
   END_VAR
BEGIN

REGION Network 2: TE102a
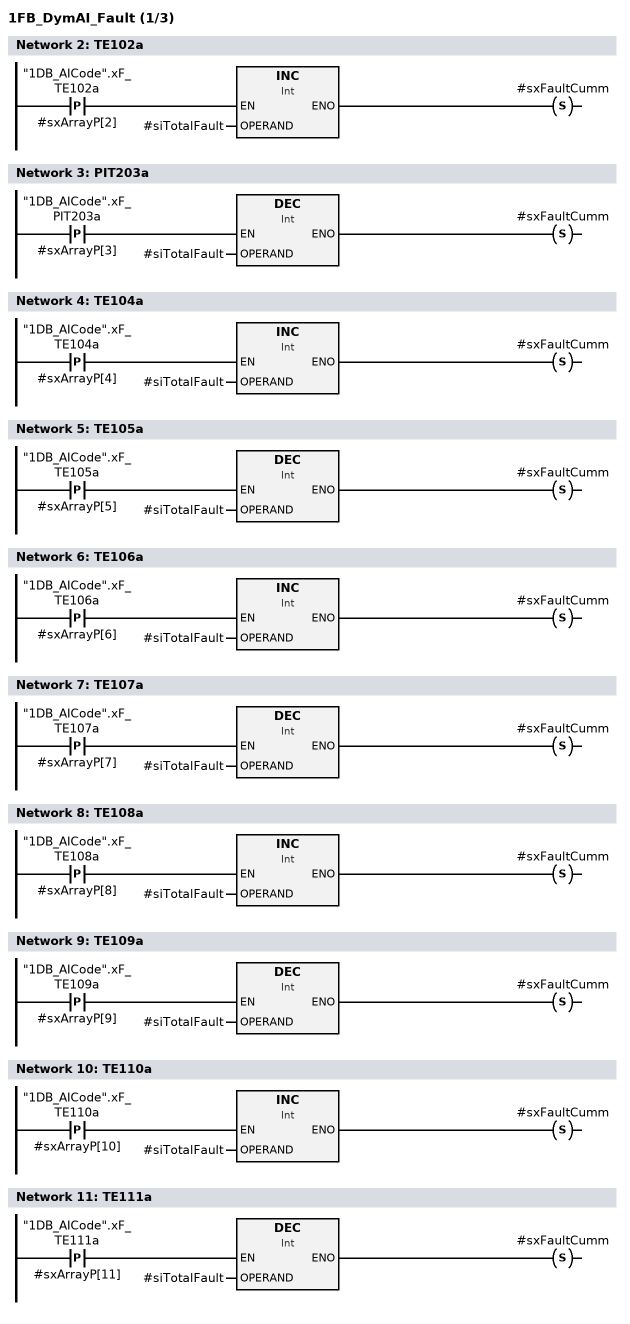
   RUNG wire#powerrail
      P_Contact(operand := "1DB_AICode".xF_TE102a, bit := #sxArrayP[2])
      { S7_Templates := "DestType := Int" } Inc( #siTotalFault )
      S_Coil( #sxFaultCumm )
   END_RUNG
   // the same network as SCL:
   #_w1 := "1DB_AICode".xF_TE102a AND NOT #sxArrayP[2];   // rising edge of "1DB_AICode".xF_TE102a
   #sxArrayP[2] := "1DB_AICode".xF_TE102a;
   IF #_w1 THEN
       #siTotalFault := #siTotalFault + 1;
       #sxFaultCumm := TRUE;
   END_IF;
END_REGION

REGION Network 3: PIT203a
   RUNG wire#powerrail
      P_Contact(operand := "1DB_AICode".xF_PIT203a, bit := #sxArrayP[3])
      { S7_Templates := "DestType := Int" } Dec( #siTotalFault )
      S_Coil( #sxFaultCumm )
   END_RUNG
   // the same network as SCL:
   #_w1 := "1DB_AICode".xF_PIT203a AND NOT #sxArrayP[3];   // rising edge of "1DB_AICode".xF_PIT203a
   #sxArrayP[3] := "1DB_AICode".xF_PIT203a;
   IF #_w1 THEN
       #siTotalFault := #siTotalFault - 1;
       #sxFaultCumm := TRUE;
   END_IF;
END_REGION

REGION Network 4: TE104a
   RUNG wire#powerrail
      P_Contact(operand := "1DB_AICode".xF_TE104a, bit := #sxArrayP[4])
      { S7_Templates := "DestType := Int" } Inc( #siTotalFault )
      S_Coil( #sxFaultCumm )
   END_RUNG
   // the same network as SCL:
   #_w1 := "1DB_AICode".xF_TE104a AND NOT #sxArrayP[4];   // rising edge of "1DB_AICode".xF_TE104a
   #sxArrayP[4] := "1DB_AICode".xF_TE104a;
   IF #_w1 THEN
       #siTotalFault := #siTotalFault + 1;
       #sxFaultCumm := TRUE;
   END_IF;
END_REGION

REGION Network 5: TE105a
   RUNG wire#powerrail
      P_Contact(operand := "1DB_AICode".xF_TE105a, bit := #sxArrayP[5])
      { S7_Templates := "DestType := Int" } Dec( #siTotalFault )
      S_Coil( #sxFaultCumm )
   END_RUNG
   // the same network as SCL:
   #_w1 := "1DB_AICode".xF_TE105a AND NOT #sxArrayP[5];   // rising edge of "1DB_AICode".xF_TE105a
   #sxArrayP[5] := "1DB_AICode".xF_TE105a;
   IF #_w1 THEN
       #siTotalFault := #siTotalFault - 1;
       #sxFaultCumm := TRUE;
   END_IF;
END_REGION

REGION Network 6: TE106a
   RUNG wire#powerrail
      P_Contact(operand := "1DB_AICode".xF_TE106a, bit := #sxArrayP[6])
      { S7_Templates := "DestType := Int" } Inc( #siTotalFault )
      S_Coil( #sxFaultCumm )
   END_RUNG
   // the same network as SCL:
   #_w1 := "1DB_AICode".xF_TE106a AND NOT #sxArrayP[6];   // rising edge of "1DB_AICode".xF_TE106a
   #sxArrayP[6] := "1DB_AICode".xF_TE106a;
   IF #_w1 THEN
       #siTotalFault := #siTotalFault + 1;
       #sxFaultCumm := TRUE;
   END_IF;
END_REGION

REGION Network 7: TE107a
   RUNG wire#powerrail
      P_Contact(operand := "1DB_AICode".xF_TE107a, bit := #sxArrayP[7])
      { S7_Templates := "DestType := Int" } Dec( #siTotalFault )
      S_Coil( #sxFaultCumm )
   END_RUNG
   // the same network as SCL:
   #_w1 := "1DB_AICode".xF_TE107a AND NOT #sxArrayP[7];   // rising edge of "1DB_AICode".xF_TE107a
   #sxArrayP[7] := "1DB_AICode".xF_TE107a;
   IF #_w1 THEN
       #siTotalFault := #siTotalFault - 1;
       #sxFaultCumm := TRUE;
   END_IF;
END_REGION

REGION Network 8: TE108a
   RUNG wire#powerrail
      P_Contact(operand := "1DB_AICode".xF_TE108a, bit := #sxArrayP[8])
      { S7_Templates := "DestType := Int" } Inc( #siTotalFault )
      S_Coil( #sxFaultCumm )
   END_RUNG
   // the same network as SCL:
   #_w1 := "1DB_AICode".xF_TE108a AND NOT #sxArrayP[8];   // rising edge of "1DB_AICode".xF_TE108a
   #sxArrayP[8] := "1DB_AICode".xF_TE108a;
   IF #_w1 THEN
       #siTotalFault := #siTotalFault + 1;
       #sxFaultCumm := TRUE;
   END_IF;
END_REGION

REGION Network 9: TE109a
   RUNG wire#powerrail
      P_Contact(operand := "1DB_AICode".xF_TE109a, bit := #sxArrayP[9])
      { S7_Templates := "DestType := Int" } Dec( #siTotalFault )
      S_Coil( #sxFaultCumm )
   END_RUNG
   // the same network as SCL:
   #_w1 := "1DB_AICode".xF_TE109a AND NOT #sxArrayP[9];   // rising edge of "1DB_AICode".xF_TE109a
   #sxArrayP[9] := "1DB_AICode".xF_TE109a;
   IF #_w1 THEN
       #siTotalFault := #siTotalFault - 1;
       #sxFaultCumm := TRUE;
   END_IF;
END_REGION

REGION Network 10: TE110a
   RUNG wire#powerrail
      P_Contact(operand := "1DB_AICode".xF_TE110a, bit := #sxArrayP[10])
      { S7_Templates := "DestType := Int" } Inc( #siTotalFault )
      S_Coil( #sxFaultCumm )
   END_RUNG
   // the same network as SCL:
   #_w1 := "1DB_AICode".xF_TE110a AND NOT #sxArrayP[10];   // rising edge of "1DB_AICode".xF_TE110a
   #sxArrayP[10] := "1DB_AICode".xF_TE110a;
   IF #_w1 THEN
       #siTotalFault := #siTotalFault + 1;
       #sxFaultCumm := TRUE;
   END_IF;
END_REGION

REGION Network 11: TE111a
   RUNG wire#powerrail
      P_Contact(operand := "1DB_AICode".xF_TE111a, bit := #sxArrayP[11])
      { S7_Templates := "DestType := Int" } Dec( #siTotalFault )
      S_Coil( #sxFaultCumm )
   END_RUNG
   // the same network as SCL:
   #_w1 := "1DB_AICode".xF_TE111a AND NOT #sxArrayP[11];   // rising edge of "1DB_AICode".xF_TE111a
   #sxArrayP[11] := "1DB_AICode".xF_TE111a;
   IF #_w1 THEN
       #siTotalFault := #siTotalFault - 1;
       #sxFaultCumm := TRUE;
   END_IF;
END_REGION

REGION Network 12: TE112a
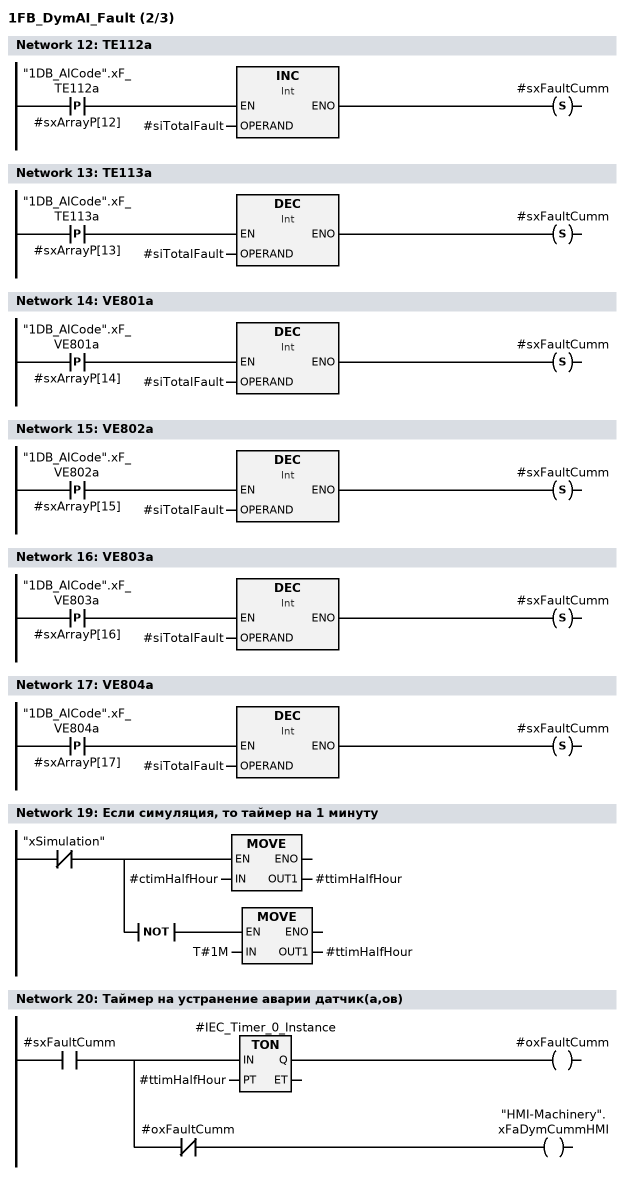
   RUNG wire#powerrail
      P_Contact(operand := "1DB_AICode".xF_TE112a, bit := #sxArrayP[12])
      { S7_Templates := "DestType := Int" } Inc( #siTotalFault )
      S_Coil( #sxFaultCumm )
   END_RUNG
   // the same network as SCL:
   #_w1 := "1DB_AICode".xF_TE112a AND NOT #sxArrayP[12];   // rising edge of "1DB_AICode".xF_TE112a
   #sxArrayP[12] := "1DB_AICode".xF_TE112a;
   IF #_w1 THEN
       #siTotalFault := #siTotalFault + 1;
       #sxFaultCumm := TRUE;
   END_IF;
END_REGION

REGION Network 13: TE113a
   RUNG wire#powerrail
      P_Contact(operand := "1DB_AICode".xF_TE113a, bit := #sxArrayP[13])
      { S7_Templates := "DestType := Int" } Dec( #siTotalFault )
      S_Coil( #sxFaultCumm )
   END_RUNG
   // the same network as SCL:
   #_w1 := "1DB_AICode".xF_TE113a AND NOT #sxArrayP[13];   // rising edge of "1DB_AICode".xF_TE113a
   #sxArrayP[13] := "1DB_AICode".xF_TE113a;
   IF #_w1 THEN
       #siTotalFault := #siTotalFault - 1;
       #sxFaultCumm := TRUE;
   END_IF;
END_REGION

REGION Network 14: VE801a
   RUNG wire#powerrail
      P_Contact(operand := "1DB_AICode".xF_VE801a, bit := #sxArrayP[14])
      { S7_Templates := "DestType := Int" } Dec( #siTotalFault )
      S_Coil( #sxFaultCumm )
   END_RUNG
   // the same network as SCL:
   #_w1 := "1DB_AICode".xF_VE801a AND NOT #sxArrayP[14];   // rising edge of "1DB_AICode".xF_VE801a
   #sxArrayP[14] := "1DB_AICode".xF_VE801a;
   IF #_w1 THEN
       #siTotalFault := #siTotalFault - 1;
       #sxFaultCumm := TRUE;
   END_IF;
END_REGION

REGION Network 15: VE802a
   RUNG wire#powerrail
      P_Contact(operand := "1DB_AICode".xF_VE802a, bit := #sxArrayP[15])
      { S7_Templates := "DestType := Int" } Dec( #siTotalFault )
      S_Coil( #sxFaultCumm )
   END_RUNG
   // the same network as SCL:
   #_w1 := "1DB_AICode".xF_VE802a AND NOT #sxArrayP[15];   // rising edge of "1DB_AICode".xF_VE802a
   #sxArrayP[15] := "1DB_AICode".xF_VE802a;
   IF #_w1 THEN
       #siTotalFault := #siTotalFault - 1;
       #sxFaultCumm := TRUE;
   END_IF;
END_REGION

REGION Network 16: VE803a
   RUNG wire#powerrail
      P_Contact(operand := "1DB_AICode".xF_VE803a, bit := #sxArrayP[16])
      { S7_Templates := "DestType := Int" } Dec( #siTotalFault )
      S_Coil( #sxFaultCumm )
   END_RUNG
   // the same network as SCL:
   #_w1 := "1DB_AICode".xF_VE803a AND NOT #sxArrayP[16];   // rising edge of "1DB_AICode".xF_VE803a
   #sxArrayP[16] := "1DB_AICode".xF_VE803a;
   IF #_w1 THEN
       #siTotalFault := #siTotalFault - 1;
       #sxFaultCumm := TRUE;
   END_IF;
END_REGION

REGION Network 17: VE804a
   RUNG wire#powerrail
      P_Contact(operand := "1DB_AICode".xF_VE804a, bit := #sxArrayP[17])
      { S7_Templates := "DestType := Int" } Dec( #siTotalFault )
      S_Coil( #sxFaultCumm )
   END_RUNG
   // the same network as SCL:
   #_w1 := "1DB_AICode".xF_VE804a AND NOT #sxArrayP[17];   // rising edge of "1DB_AICode".xF_VE804a
   #sxArrayP[17] := "1DB_AICode".xF_VE804a;
   IF #_w1 THEN
       #siTotalFault := #siTotalFault - 1;
       #sxFaultCumm := TRUE;
   END_IF;
END_REGION

REGION Network 18: Авария от ШПЧ1 (перенесено в сигнализацию)
END_REGION

REGION Network 19: Если симуляция, то таймер на 1 минуту
   RUNG wire#powerrail
      I_Contact( "xSimulation" )
      wire#w1
      Move(in := #ctimHalfHour, out1 => #ttimHalfHour)
   END_RUNG
   RUNG wire#w1
      Not()
      Move(in := T#1M, out1 => #ttimHalfHour)
   END_RUNG
   // the same network as SCL:
   IF NOT "xSimulation" THEN #ttimHalfHour := #ctimHalfHour; END_IF;
   IF NOT (NOT "xSimulation") THEN #ttimHalfHour := T#1M; END_IF;
END_REGION

REGION Network 20: Таймер на устранение аварии датчик(а,ов)
   #IEC_Timer_0_Instance(IN := #sxFaultCumm, PT := #ttimHalfHour);   // TON
   #oxFaultCumm := #IEC_Timer_0_Instance.Q;
   "HMI-Machinery".xFaDymCummHMI := #sxFaultCumm AND NOT #oxFaultCumm;
END_REGION

REGION Network 21: Таймер обратного отсчета
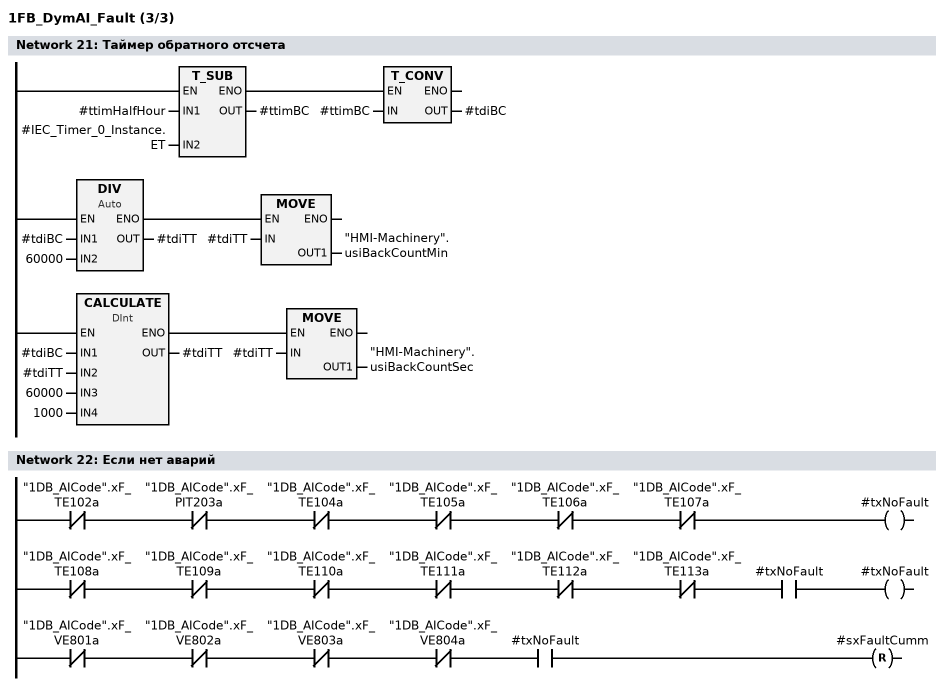
   // ENO of a box is taken as its EN; it also drops when the box reports an error
   #ttimBC := T_SUB(IN1 := #ttimHalfHour, IN2 := #IEC_Timer_0_Instance.ET);
   #tdiBC := T_CONV(IN := #ttimBC);
   #tdiTT := #tdiBC / 60000;
   "HMI-Machinery".usiBackCountMin := #tdiTT;
   #tdiTT := (#tdiBC - (#tdiTT * 60000)) / 1000;
   "HMI-Machinery".usiBackCountSec := #tdiTT;
END_REGION

REGION Network 22: Если нет аварий
   RUNG wire#powerrail
      I_Contact( "1DB_AICode".xF_TE102a )
      I_Contact( "1DB_AICode".xF_PIT203a )
      I_Contact( "1DB_AICode".xF_TE104a )
      I_Contact( "1DB_AICode".xF_TE105a )
      I_Contact( "1DB_AICode".xF_TE106a )
      I_Contact( "1DB_AICode".xF_TE107a )
      Coil( #txNoFault )
   END_RUNG
   RUNG wire#powerrail
      I_Contact( "1DB_AICode".xF_TE108a )
      I_Contact( "1DB_AICode".xF_TE109a )
      I_Contact( "1DB_AICode".xF_TE110a )
      I_Contact( "1DB_AICode".xF_TE111a )
      I_Contact( "1DB_AICode".xF_TE112a )
      I_Contact( "1DB_AICode".xF_TE113a )
      Contact( #txNoFault )
      Coil( #txNoFault )
   END_RUNG
   RUNG wire#powerrail
      I_Contact( "1DB_AICode".xF_VE801a )
      I_Contact( "1DB_AICode".xF_VE802a )
      I_Contact( "1DB_AICode".xF_VE803a )
      I_Contact( "1DB_AICode".xF_VE804a )
      Contact( #txNoFault )
      R_Coil( #sxFaultCumm )
   END_RUNG
   // the same network as SCL:
   #txNoFault := NOT "1DB_AICode".xF_TE102a AND NOT "1DB_AICode".xF_PIT203a AND NOT "1DB_AICode".xF_TE104a AND NOT "1DB_AICode".xF_TE105a AND NOT "1DB_AICode".xF_TE106a AND NOT "1DB_AICode".xF_TE107a;
   #txNoFault := NOT "1DB_AICode".xF_TE108a AND NOT "1DB_AICode".xF_TE109a AND NOT "1DB_AICode".xF_TE110a AND NOT "1DB_AICode".xF_TE111a AND NOT "1DB_AICode".xF_TE112a AND NOT "1DB_AICode".xF_TE113a AND #txNoFault;
   IF NOT "1DB_AICode".xF_VE801a AND NOT "1DB_AICode".xF_VE802a AND NOT "1DB_AICode".xF_VE803a AND NOT "1DB_AICode".xF_VE804a AND #txNoFault THEN
       #sxFaultCumm := FALSE;
   END_IF;
END_REGION
END_FUNCTION_BLOCK

FUNCTION "1FC_DymRestart" : Void   // FC99, LAD
{ S7_Optimized_Access := 'TRUE' }
VERSION : 0.1
   VAR_INPUT
      itim150 : Time;   // Время запрета повторного старта
   END_VAR
   VAR_TEMP
      ttimBC : Time;   // Обратный отсчет в формате Time
      tdiBC : DInt;   // Сконвертированное время
      tdiTT : DInt;   // Временная переменная
   END_VAR
BEGIN

REGION Network 2: Находим разность и конвертируем
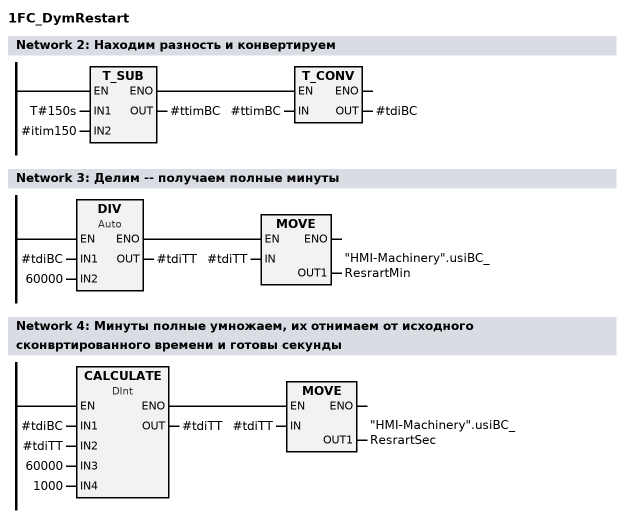
   // ENO of a box is taken as its EN; it also drops when the box reports an error
   #ttimBC := T_SUB(IN1 := T#150s, IN2 := #itim150);
   #tdiBC := T_CONV(IN := #ttimBC);
END_REGION

REGION Network 3: Делим -- получаем полные минуты
   RUNG wire#powerrail
      Div(in1 := #tdiBC, in2 := 60000, out => #tdiTT)
      Move(in := #tdiTT, out1 => "HMI-Machinery".usiBC_ResrartMin)
   END_RUNG
   // the same network as SCL:
   #tdiTT := #tdiBC / 60000;
   "HMI-Machinery".usiBC_ResrartMin := #tdiTT;
END_REGION

REGION Network 4: Минуты полные умножаем, их отнимаем от исходного сконвртированного времени и готовы секунды
   RUNG wire#powerrail
      { S7_Templates := "SrcType := DInt"; S7_Expression := "(IN1 - (IN2 * IN3)) / IN4" } Calculate(in1 := #tdiBC, in2 := #tdiTT, in3 := 60000, in4 := 1000, out => #tdiTT)
      Move(in := #tdiTT, out1 => "HMI-Machinery".usiBC_ResrartSec)
   END_RUNG
   // the same network as SCL:
   #tdiTT := (#tdiBC - (#tdiTT * 60000)) / 1000;
   "HMI-Machinery".usiBC_ResrartSec := #tdiTT;
END_REGION
END_FUNCTION

ORGANIZATION_BLOCK "Time error interrupt"   // OB80, LAD, TimeErrorInterrupt
{ S7_Optimized_Access := 'TRUE' }
VERSION : 0.1
   VAR_INPUT
      Fault_ID : Byte;   // Fault identifier
      Csg_OBnr : OB_Any;   // Number of OB causing the error
      Csg_Prio : UInt;   // Priority of OB causing the error
   END_VAR
BEGIN
END_ORGANIZATION_BLOCK

ORGANIZATION_BLOCK "Diagnostic error interrupt"   // OB82, LAD, DiagnosticErrorInterrupt
{ S7_Optimized_Access := 'TRUE' }
VERSION : 0.1
   VAR_INPUT
      IO_State : Word;   // IO state of the HW object
      LADDR : Hw_Any;   // Hardware identifier
      Channel : UInt;   // Channel number
      MultiError : Bool;   // =true if more than one error is present
   END_VAR
BEGIN
END_ORGANIZATION_BLOCK

ORGANIZATION_BLOCK "Pull or plug of modules"   // OB83, LAD, PullPlug
{ S7_Optimized_Access := 'TRUE' }
VERSION : 0.1
   VAR_INPUT
      LADDR : Hw_Io;   // Hardware identifier
      Event_Class : Byte;   // 16#38/39: module inserted, removed
      Fault_ID : Byte;   // Fault identifier
   END_VAR
BEGIN
END_ORGANIZATION_BLOCK

ORGANIZATION_BLOCK "Rack or station failure"   // OB86, LAD, RackStationFailure
{ S7_Optimized_Access := 'TRUE' }
VERSION : 0.1
   VAR_INPUT
      LADDR : Hw_Device;   // Hardware identifier
      Event_Class : Byte;   // Event class
      Fault_ID : Byte;   // Fault identifier
   END_VAR
BEGIN
END_ORGANIZATION_BLOCK

// folder: Machinery

FUNCTION_BLOCK "1FB_CommTest"   // FB98, LAD
{ S7_Optimized_Access := 'TRUE' }
VERSION : 0.1
   VAR
      sxForFront : Bool;   // Определение фронта
      sxStart2 : Bool;   // Импульсы один раз на 2сек
      IEC_Timer_0_Instance : TP_TIME;
      swCounterOld : UInt;   // Старое значение счетчика в ПЛК1
   END_VAR
   VAR_TEMP   // added for the SCL form of the ladder/FBD networks
      _w1 : Bool;
   END_VAR
BEGIN

REGION Network 2: Инкремент счетчика для ПЛК1
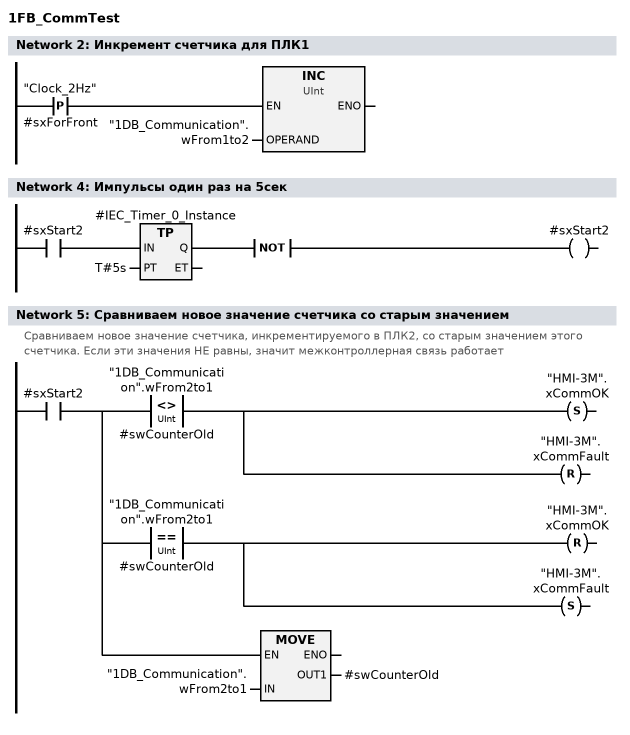
   RUNG wire#powerrail
      P_Contact(operand := "Clock_2Hz", bit := #sxForFront)
      { S7_Templates := "DestType := UInt" } Inc( "1DB_Communication".wFrom1to2 )
   END_RUNG
   // the same network as SCL:
   #_w1 := "Clock_2Hz" AND NOT #sxForFront;   // rising edge of "Clock_2Hz"
   #sxForFront := "Clock_2Hz";
   IF #_w1 THEN "1DB_Communication".wFrom1to2 := "1DB_Communication".wFrom1to2 + 1; END_IF;
END_REGION

REGION Network 4: Импульсы один раз на 5сек
   #IEC_Timer_0_Instance(IN := #sxStart2, PT := T#5s);   // TP
   #sxStart2 := NOT #IEC_Timer_0_Instance.Q;
END_REGION

REGION Network 5: Сравниваем новое значение счетчика со старым значением
   // Сравниваем новое значение счетчика, инкрементируемого в ПЛК2, со старым значением этого счетчика. Если эти значения НЕ равны, значит межконтроллерная связь работает
   RUNG wire#powerrail
      Contact( #sxStart2 )
      wire#w1
      { S7_Templates := "SrcType := UInt" } NE_Contact(in1 := "1DB_Communication".wFrom2to1, in2 := #swCounterOld)
      wire#w2
      S_Coil( "HMI-3M".xCommOK )
   END_RUNG
   RUNG wire#w2
      R_Coil( "HMI-3M".xCommFault )
   END_RUNG
   RUNG wire#w1
      { S7_Templates := "SrcType := UInt" } EQ_Contact(in1 := "1DB_Communication".wFrom2to1, in2 := #swCounterOld)
      wire#w3
      R_Coil( "HMI-3M".xCommOK )
   END_RUNG
   RUNG wire#w3
      S_Coil( "HMI-3M".xCommFault )
   END_RUNG
   RUNG wire#w1
      Move(in := "1DB_Communication".wFrom2to1, out1 => #swCounterOld)
   END_RUNG
   // the same network as SCL:
   IF #sxStart2 AND ("1DB_Communication".wFrom2to1 <> #swCounterOld) THEN
       "HMI-3M".xCommOK := TRUE;
       "HMI-3M".xCommFault := FALSE;
   END_IF;
   IF #sxStart2 AND ("1DB_Communication".wFrom2to1 = #swCounterOld) THEN
       "HMI-3M".xCommOK := FALSE;
       "HMI-3M".xCommFault := TRUE;
   END_IF;
   IF #sxStart2 THEN #swCounterOld := "1DB_Communication".wFrom2to1; END_IF;
END_REGION
END_FUNCTION_BLOCK

FUNCTION_BLOCK "Control1M"   // FB501, LAD
TITLE = Управление Регулирующим клапаном 1М
{ S7_Optimized_Access := 'TRUE' }
VERSION : 0.1
   VAR_INPUT
      irPosition : Real;   // Положение механизма
      ixMEO_Ready : Bool;   // Готовность МЭО
      ixFullOpen : Bool;   // Полностью открыт
      ixFullClose : Bool;   // Полностью закрыт
      ixRemoteContr : Bool;   // Ключ в положении Дистанционный рехим
      ixExtStop : Bool;   // Внешняя блокировка
      ixExtFullOpen : Bool;   // Внешняя команда на полное открытие
   END_VAR
   VAR_OUTPUT
      oxButMore : Bool;   // Кнопка на ручное открытие
      oxButLess : Bool;   // Кнопка на ручное закрытие
      orPosGoTo : Real;   // Уставка перемещения в заданное положение [%]
      oxButGoTo : Bool;   // Кнопка Перемещение В Заданное Положение
      oxSwitchAutoMode : Bool;   // Переключатель (автомат.=1, ручной=0) на ЧМИ
      oxReady : Bool;   // Готовность механизма
      oxCommandOpen : Bool;   // Команда на открытие
      oxCommandClose : Bool;   // Команда на закрытие
   END_VAR
   VAR_IN_OUT
      "ioHMI-M" : "uHMI-Machine";   // Структура данных связи с ЧМИ
   END_VAR
   VAR
      sxWarning : Bool;   // Есть предупреждения
      sxFault : Bool;   // Есть авария
      sxWork : Bool;   // Есть моя команда
      sxForF1 : Bool;   // Бит для определения фронта
      sxForF2 : Bool;   // Бит для определения фронта
      sxForF3 : Bool;   // Бит для определения фронта
      sxForF4 : Bool;   // Бит для определения фронта
      sxForF5 : Bool;   // Бит для определения фронта
      IEC_Timer_0_Instance : TON_TIME;   // Таймер
      srPosOld : Real;   // Старое значение позиции
      sxWorkOld : Bool;   // Бит старого значения sxWork
      sxGoTo : Bool;   // Бит Перемещения В Заданую Позицию
      sb1000 : Byte;   // Проверка секундного импульса
      sb1001 : Byte;   // Проверка секундного импульса
      sb1002 : Byte;   // Проверка секундного импульса
      ssStatus : String;
   END_VAR
   VAR_TEMP
      tr1 : Real;   // Временный риэл
      tx1 : Bool;   // Временный бит
      tx2 : Bool;   // Временный бит
   END_VAR
   VAR CONSTANT
      c10 : String := 'Ready';
      c20 : String := 'Not ready';
      c30 : String := 'Fault';
      c40 : String := 'External lock';
   END_VAR
   VAR_TEMP   // added for the SCL form of the ladder/FBD networks
      _w1 : Bool;
      _w2 : Bool;
      _w3 : Bool;
      _w4 : Bool;
   END_VAR
BEGIN

REGION Network 1: Подготовка данных для HMI:
END_REGION

REGION Network 2: -положение клапана
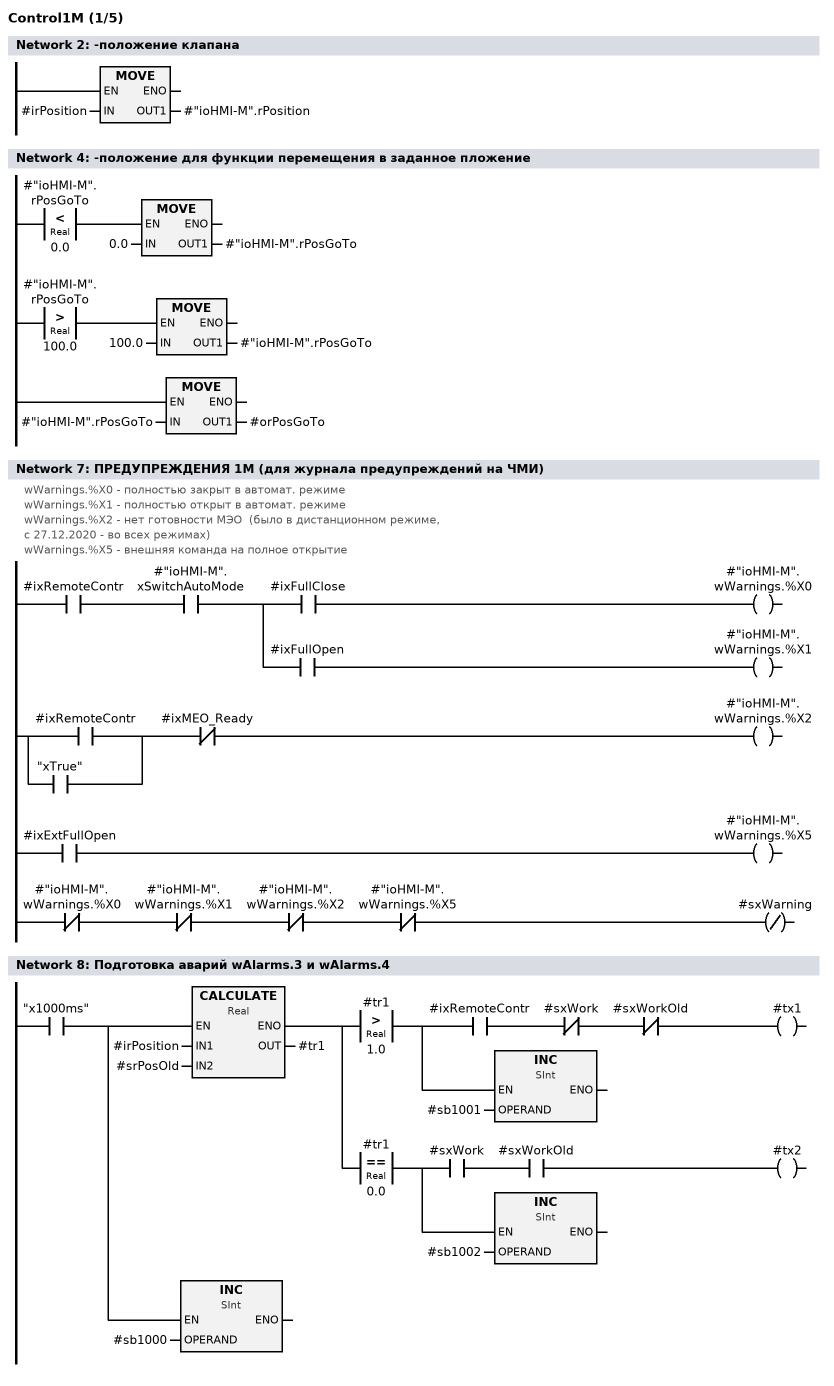
   RUNG wire#powerrail
      Move(in := #irPosition, out1 => #"ioHMI-M".rPosition)
   END_RUNG
   // the same network as SCL:
   #"ioHMI-M".rPosition := #irPosition;
END_REGION

REGION Network 3: Подготовка данных от HMI:
END_REGION

REGION Network 4: -положение для функции перемещения в заданное пложение
   RUNG wire#powerrail
      { S7_Templates := "SrcType := Real" } LT_Contact(in1 := #"ioHMI-M".rPosGoTo, in2 := 0.0)
      Move(in := 0.0, out1 => #"ioHMI-M".rPosGoTo)
   END_RUNG
   RUNG wire#powerrail
      { S7_Templates := "SrcType := Real" } GT_Contact(in1 := #"ioHMI-M".rPosGoTo, in2 := 100.0)
      Move(in := 100.0, out1 => #"ioHMI-M".rPosGoTo)
   END_RUNG
   RUNG wire#powerrail
      Move(in := #"ioHMI-M".rPosGoTo, out1 => #orPosGoTo)
   END_RUNG
   // the same network as SCL:
   IF #"ioHMI-M".rPosGoTo < 0.0 THEN #"ioHMI-M".rPosGoTo := 0.0; END_IF;
   IF #"ioHMI-M".rPosGoTo > 100.0 THEN #"ioHMI-M".rPosGoTo := 100.0; END_IF;
   #orPosGoTo := #"ioHMI-M".rPosGoTo;
END_REGION

REGION Network 5 (SCL): -кнопки на ЧМИ
   #oxButMore  :=  #"ioHMI-M".xButManOpen;
   #oxButLess  :=  #"ioHMI-M".xButManClose;
   #oxButGoTo  :=  #"ioHMI-M".xButtonGoTo;
   #oxSwitchAutoMode := #"ioHMI-M".xSwitchAutoMode;
END_REGION

REGION Network 7: ПРЕДУПРЕЖДЕНИЯ 1М (для журнала предупреждений на ЧМИ)
   // wWarnings.%X0 - полностью закрыт в автомат. режиме
   // wWarnings.%X1 - полностью открыт в автомат. режиме
   // wWarnings.%X2 - нет готовности МЭО  (было в дистанционном режиме, 
   //                                с 27.12.2020 - во всех режимах)
   // wWarnings.%X5 - внешняя команда на полное открытие
   RUNG wire#powerrail
      Contact( #ixRemoteContr )
      Contact( #"ioHMI-M".xSwitchAutoMode )
      wire#w1
      Contact( #ixFullClose )
      Coil( #"ioHMI-M".wWarnings.%X0 )
   END_RUNG
   RUNG wire#w1
      Contact( #ixFullOpen )
      Coil( #"ioHMI-M".wWarnings.%X1 )
   END_RUNG
   RUNG wire#powerrail
      Contact( #ixRemoteContr )
      wire#w2
      I_Contact( #ixMEO_Ready )
      Coil( #"ioHMI-M".wWarnings.%X2 )
   END_RUNG
   RUNG wire#powerrail
      Contact( "xTrue" )
   END_RUNG wire#w2
   RUNG wire#powerrail
      Contact( #ixExtFullOpen )
      Coil( #"ioHMI-M".wWarnings.%X5 )
   END_RUNG
   RUNG wire#powerrail
      I_Contact( #"ioHMI-M".wWarnings.%X0 )
      I_Contact( #"ioHMI-M".wWarnings.%X1 )
      I_Contact( #"ioHMI-M".wWarnings.%X2 )
      I_Contact( #"ioHMI-M".wWarnings.%X5 )
      I_Coil( #sxWarning )
   END_RUNG
   // the same network as SCL:
   #_w1 := #ixRemoteContr AND #"ioHMI-M".xSwitchAutoMode;
   #"ioHMI-M".wWarnings.%X0 := #_w1 AND #ixFullClose;
   #"ioHMI-M".wWarnings.%X1 := #_w1 AND #ixFullOpen;
   #"ioHMI-M".wWarnings.%X2 := (#ixRemoteContr OR "xTrue") AND NOT #ixMEO_Ready;
   #"ioHMI-M".wWarnings.%X5 := #ixExtFullOpen;
   #sxWarning := NOT (NOT #"ioHMI-M".wWarnings.%X0 AND NOT #"ioHMI-M".wWarnings.%X1 AND NOT #"ioHMI-M".wWarnings.%X2 AND NOT #"ioHMI-M".wWarnings.%X5);
END_REGION

REGION Network 8: Подготовка аварий wAlarms.3 и wAlarms.4
   RUNG wire#powerrail
      Contact( "x1000ms" )
      wire#w1
      { S7_Templates := "SrcType := Real"; S7_Expression := "ABS(IN1-IN2)" } Calculate(in1 := #irPosition, in2 := #srPosOld, out => #tr1)
      wire#w2
      { S7_Templates := "SrcType := Real" } GT_Contact(in1 := #tr1, in2 := 1.0)
      wire#w3
      Contact( #ixRemoteContr )
      I_Contact( #sxWork )
      I_Contact( #sxWorkOld )
      Coil( #tx1 )
   END_RUNG
   RUNG wire#w3
      { S7_Templates := "DestType := SInt" } Inc( #sb1001 )
   END_RUNG
   RUNG wire#w2
      { S7_Templates := "SrcType := Real" } EQ_Contact(in1 := #tr1, in2 := 0.0)
      wire#w4
      Contact( #sxWork )
      Contact( #sxWorkOld )
      Coil( #tx2 )
   END_RUNG
   RUNG wire#w4
      { S7_Templates := "DestType := SInt" } Inc( #sb1002 )
   END_RUNG
   RUNG wire#w1
      { S7_Templates := "DestType := SInt" } Inc( #sb1000 )
   END_RUNG
   // the same network as SCL:
   IF "x1000ms" THEN #tr1 := ABS(#irPosition-#srPosOld); END_IF;
   #_w1 := "x1000ms" AND (#tr1 > 1.0);
   #tx1 := #_w1 AND #ixRemoteContr AND NOT #sxWork AND NOT #sxWorkOld;
   IF #_w1 THEN #sb1001 := #sb1001 + 1; END_IF;
   #_w2 := "x1000ms" AND (#tr1 = 0.0);
   #tx2 := #_w2 AND #sxWork AND #sxWorkOld;
   IF #_w2 THEN #sb1002 := #sb1002 + 1; END_IF;
   IF "x1000ms" THEN #sb1000 := #sb1000 + 1; END_IF;
END_REGION

REGION Network 9: Подготовка аварий wAlarms.3 и wAlarms.4. Бит старого значения позиции #sxWork
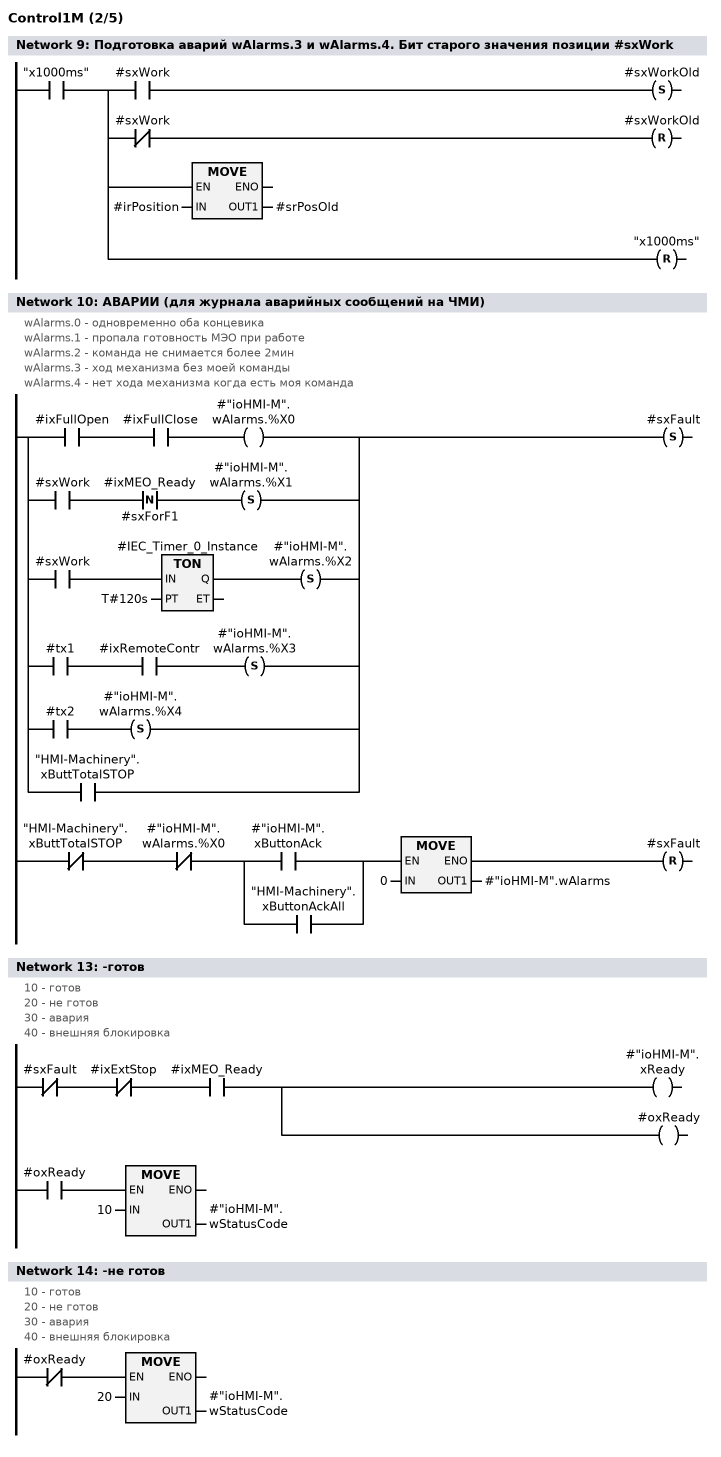
   RUNG wire#powerrail
      Contact( "x1000ms" )
      wire#w1
      Contact( #sxWork )
      S_Coil( #sxWorkOld )
   END_RUNG
   RUNG wire#w1
      I_Contact( #sxWork )
      R_Coil( #sxWorkOld )
   END_RUNG
   RUNG wire#w1
      Move(in := #irPosition, out1 => #srPosOld)
   END_RUNG
   RUNG wire#w1
      R_Coil( "x1000ms" )
   END_RUNG
   // the same network as SCL:
   IF "x1000ms" AND #sxWork THEN #sxWorkOld := TRUE; END_IF;
   IF "x1000ms" AND NOT #sxWork THEN #sxWorkOld := FALSE; END_IF;
   IF "x1000ms" THEN
       #srPosOld := #irPosition;
       "x1000ms" := FALSE;
   END_IF;
END_REGION

REGION Network 10: АВАРИИ (для журнала аварийных сообщений на ЧМИ)
   // wAlarms.0 - одновременно оба концевика
   // wAlarms.1 - пропала готовность МЭО при работе
   // wAlarms.2 - команда не снимается более 2мин
   // wAlarms.3 - ход механизма без моей команды 
   // wAlarms.4 - нет хода механизма когда есть моя команда
   #"ioHMI-M".wAlarms.%X0 := #ixFullOpen AND #ixFullClose;
   #_w1 := #sxWork AND NOT #ixMEO_Ready AND #sxForF1;   // falling edge of #ixMEO_Ready
   #sxForF1 := #ixMEO_Ready;
   #_w2 := #"ioHMI-M".wAlarms.%X0;
   IF #_w1 THEN #"ioHMI-M".wAlarms.%X1 := TRUE; END_IF;
   #IEC_Timer_0_Instance(IN := #sxWork, PT := T#120s);   // TON
   IF #IEC_Timer_0_Instance.Q THEN #"ioHMI-M".wAlarms.%X2 := TRUE; END_IF;
   #_w3 := #tx1 AND #ixRemoteContr;
   IF #_w3 THEN #"ioHMI-M".wAlarms.%X3 := TRUE; END_IF;
   IF #tx2 THEN #"ioHMI-M".wAlarms.%X4 := TRUE; END_IF;
   IF #_w2 OR #_w1 OR #IEC_Timer_0_Instance.Q OR #_w3 OR #tx2 OR "HMI-Machinery".xButtTotalSTOP THEN
       #sxFault := TRUE;
   END_IF;
   #_w4 := NOT "HMI-Machinery".xButtTotalSTOP AND NOT #"ioHMI-M".wAlarms.%X0 AND (#"ioHMI-M".xButtonAck OR "HMI-Machinery".xButtonAckAll);
   IF #_w4 THEN
       #"ioHMI-M".wAlarms := 0;
       #sxFault := FALSE;
   END_IF;
END_REGION

REGION Network 12: Статус/состояние механизма:
END_REGION

REGION Network 13: -готов
   // 10 - готов
   // 20 - не готов
   // 30 - авария
   // 40 - внешняя блокировка
   RUNG wire#powerrail
      I_Contact( #sxFault )
      I_Contact( #ixExtStop )
      Contact( #ixMEO_Ready )
      wire#w1
      Coil( #"ioHMI-M".xReady )
   END_RUNG
   RUNG wire#w1
      Coil( #oxReady )
   END_RUNG
   RUNG wire#powerrail
      Contact( #oxReady )
      Move(in := 10, out1 => #"ioHMI-M".wStatusCode)
   END_RUNG
   // the same network as SCL:
   #"ioHMI-M".xReady := NOT #sxFault AND NOT #ixExtStop AND #ixMEO_Ready;
   #oxReady := #"ioHMI-M".xReady;
   IF #oxReady THEN #"ioHMI-M".wStatusCode := 10; END_IF;
END_REGION

REGION Network 14: -не готов
   // 10 - готов
   // 20 - не готов
   // 30 - авария
   // 40 - внешняя блокировка
   RUNG wire#powerrail
      I_Contact( #oxReady )
      Move(in := 20, out1 => #"ioHMI-M".wStatusCode)
   END_RUNG
   // the same network as SCL:
   IF NOT #oxReady THEN #"ioHMI-M".wStatusCode := 20; END_IF;
END_REGION

REGION Network 15: -авария
   // 10 - готов
   // 20 - не готов
   // 30 - авария
   // 40 - внешняя блокировка
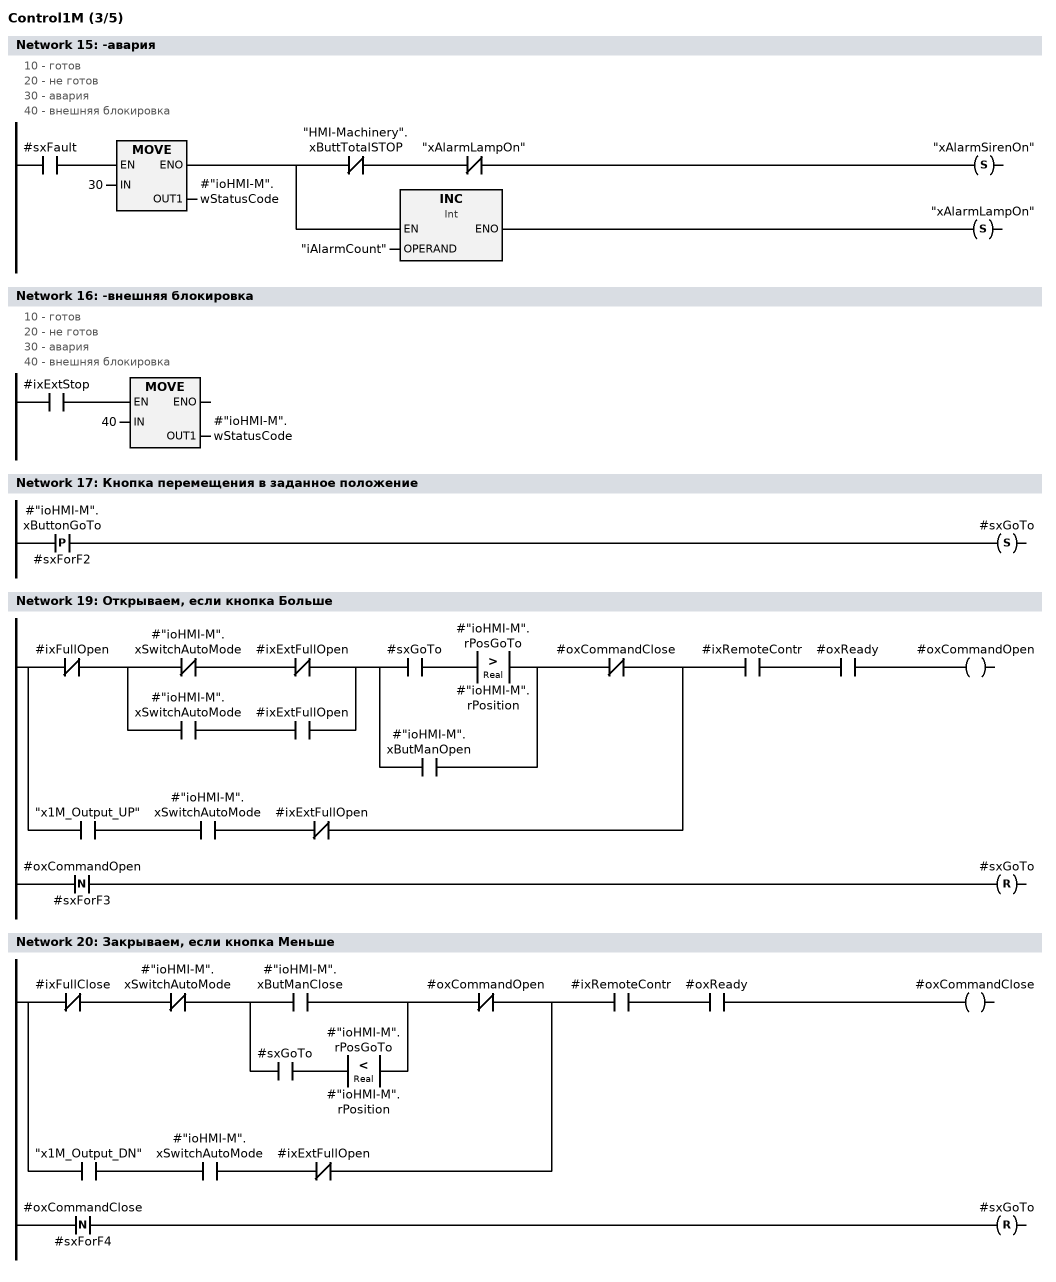
   RUNG wire#powerrail
      Contact( #sxFault )
      Move(in := 30, out1 => #"ioHMI-M".wStatusCode)
      wire#w1
      I_Contact( "HMI-Machinery".xButtTotalSTOP )
      I_Contact( "xAlarmLampOn" )
      S_Coil( "xAlarmSirenOn" )
   END_RUNG
   RUNG wire#w1
      { S7_Templates := "DestType := Int" } Inc( "iAlarmCount" )
      S_Coil( "xAlarmLampOn" )
   END_RUNG
   // the same network as SCL:
   IF #sxFault THEN #"ioHMI-M".wStatusCode := 30; END_IF;
   IF #sxFault AND NOT "HMI-Machinery".xButtTotalSTOP AND NOT "xAlarmLampOn" THEN
       "xAlarmSirenOn" := TRUE;
   END_IF;
   IF #sxFault THEN
       "iAlarmCount" := "iAlarmCount" + 1;
       "xAlarmLampOn" := TRUE;
   END_IF;
END_REGION

REGION Network 16: -внешняя блокировка
   // 10 - готов
   // 20 - не готов
   // 30 - авария
   // 40 - внешняя блокировка
   RUNG wire#powerrail
      Contact( #ixExtStop )
      Move(in := 40, out1 => #"ioHMI-M".wStatusCode)
   END_RUNG
   // the same network as SCL:
   IF #ixExtStop THEN #"ioHMI-M".wStatusCode := 40; END_IF;
END_REGION

REGION Network 17: Кнопка перемещения в заданное положение
   RUNG wire#powerrail
      P_Contact(operand := #"ioHMI-M".xButtonGoTo, bit := #sxForF2)
      S_Coil( #sxGoTo )
   END_RUNG
   // the same network as SCL:
   #_w1 := #"ioHMI-M".xButtonGoTo AND NOT #sxForF2;   // rising edge of #"ioHMI-M".xButtonGoTo
   #sxForF2 := #"ioHMI-M".xButtonGoTo;
   IF #_w1 THEN #sxGoTo := TRUE; END_IF;
END_REGION

REGION Network 18: Дистанционный РУЧНОЙ:
END_REGION

REGION Network 19: Открываем, если кнопка Больше
   RUNG wire#powerrail
      I_Contact( #ixFullOpen )
      wire#w1
      I_Contact( #"ioHMI-M".xSwitchAutoMode )
      I_Contact( #ixExtFullOpen )
      wire#w2
      Contact( #sxGoTo )
      { S7_Templates := "SrcType := Real" } GT_Contact(in1 := #"ioHMI-M".rPosGoTo, in2 := #"ioHMI-M".rPosition)
      wire#w3
      I_Contact( #oxCommandClose )
      wire#w4
      Contact( #ixRemoteContr )
      Contact( #oxReady )
      Coil( #oxCommandOpen )
   END_RUNG
   RUNG wire#w1
      Contact( #"ioHMI-M".xSwitchAutoMode )
      Contact( #ixExtFullOpen )
   END_RUNG wire#w2
   RUNG wire#w2
      Contact( #"ioHMI-M".xButManOpen )
   END_RUNG wire#w3
   RUNG wire#powerrail
      Contact( "x1M_Output_UP" )
      Contact( #"ioHMI-M".xSwitchAutoMode )
      I_Contact( #ixExtFullOpen )
   END_RUNG wire#w4
   RUNG wire#powerrail
      N_Contact(operand := #oxCommandOpen, bit := #sxForF3)
      R_Coil( #sxGoTo )
   END_RUNG
   // the same network as SCL:
   #oxCommandOpen := ((NOT #ixFullOpen AND ((NOT #"ioHMI-M".xSwitchAutoMode AND NOT #ixExtFullOpen) OR (#"ioHMI-M".xSwitchAutoMode AND #ixExtFullOpen)) AND ((#sxGoTo AND (#"ioHMI-M".rPosGoTo > #"ioHMI-M".rPosition)) OR #"ioHMI-M".xButManOpen) AND NOT #oxCommandClose) OR ("x1M_Output_UP" AND #"ioHMI-M".xSwitchAutoMode AND NOT #ixExtFullOpen)) AND #ixRemoteContr AND #oxReady;
   #_w1 := NOT #oxCommandOpen AND #sxForF3;   // falling edge of #oxCommandOpen
   #sxForF3 := #oxCommandOpen;
   IF #_w1 THEN #sxGoTo := FALSE; END_IF;
END_REGION

REGION Network 20: Закрываем, если кнопка Меньше
   RUNG wire#powerrail
      I_Contact( #ixFullClose )
      I_Contact( #"ioHMI-M".xSwitchAutoMode )
      wire#w1
      Contact( #"ioHMI-M".xButManClose )
      wire#w2
      I_Contact( #oxCommandOpen )
      wire#w3
      Contact( #ixRemoteContr )
      Contact( #oxReady )
      Coil( #oxCommandClose )
   END_RUNG
   RUNG wire#w1
      Contact( #sxGoTo )
      { S7_Templates := "SrcType := Real" } LT_Contact(in1 := #"ioHMI-M".rPosGoTo, in2 := #"ioHMI-M".rPosition)
   END_RUNG wire#w2
   RUNG wire#powerrail
      Contact( "x1M_Output_DN" )
      Contact( #"ioHMI-M".xSwitchAutoMode )
      I_Contact( #ixExtFullOpen )
   END_RUNG wire#w3
   RUNG wire#powerrail
      N_Contact(operand := #oxCommandClose, bit := #sxForF4)
      R_Coil( #sxGoTo )
   END_RUNG
   // the same network as SCL:
   #oxCommandClose := ((NOT #ixFullClose AND NOT #"ioHMI-M".xSwitchAutoMode AND (#"ioHMI-M".xButManClose OR (#sxGoTo AND (#"ioHMI-M".rPosGoTo < #"ioHMI-M".rPosition))) AND NOT #oxCommandOpen) OR ("x1M_Output_DN" AND #"ioHMI-M".xSwitchAutoMode AND NOT #ixExtFullOpen)) AND #ixRemoteContr AND #oxReady;
   #_w1 := NOT #oxCommandClose AND #sxForF4;   // falling edge of #oxCommandClose
   #sxForF4 := #oxCommandClose;
   IF #_w1 THEN #sxGoTo := FALSE; END_IF;
END_REGION

REGION Network 22: Дистанционный АВТОМАТИЧЕСКИЙ:
END_REGION

REGION Network 23: Реакция на внешний сигнал полного открытия
   // 14.01.2021 закомментирован переход в ручной режим
   // 26.01.2021 добавлено Clock_0.5Hz и переход в автомат.
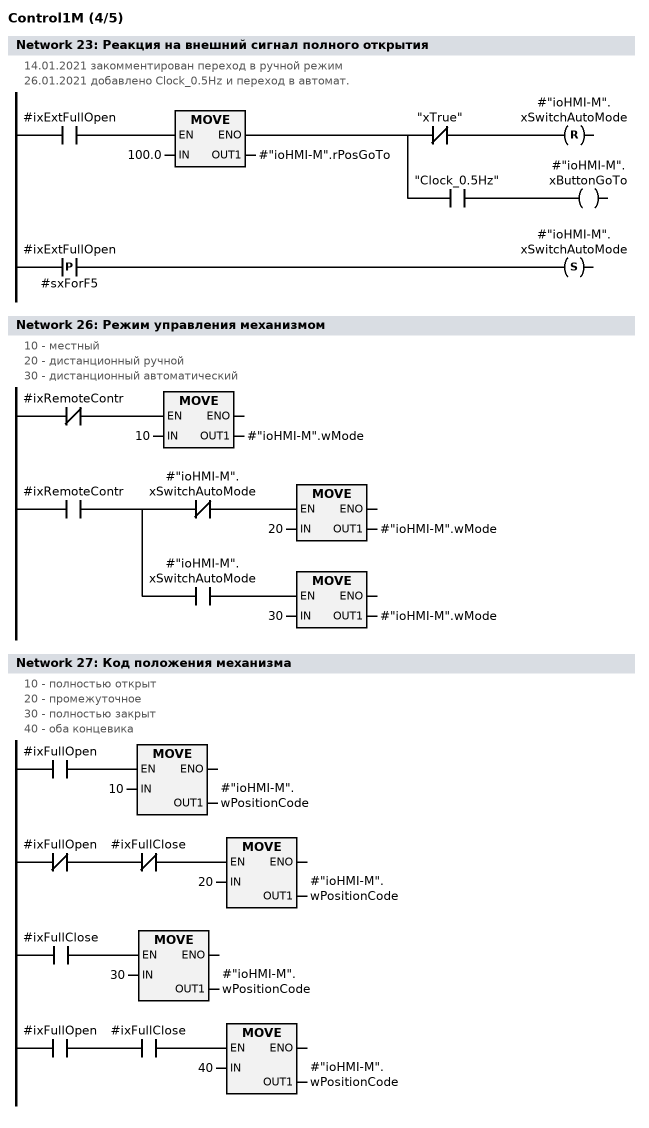
   RUNG wire#powerrail
      Contact( #ixExtFullOpen )
      Move(in := 100.0, out1 => #"ioHMI-M".rPosGoTo)
      wire#w1
      I_Contact( "xTrue" )
      R_Coil( #"ioHMI-M".xSwitchAutoMode )
   END_RUNG
   RUNG wire#w1
      Contact( "Clock_0.5Hz" )
      Coil( #"ioHMI-M".xButtonGoTo )
   END_RUNG
   RUNG wire#powerrail
      P_Contact(operand := #ixExtFullOpen, bit := #sxForF5)
      S_Coil( #"ioHMI-M".xSwitchAutoMode )
   END_RUNG
   // the same network as SCL:
   IF #ixExtFullOpen THEN #"ioHMI-M".rPosGoTo := 100.0; END_IF;
   IF #ixExtFullOpen AND NOT "xTrue" THEN #"ioHMI-M".xSwitchAutoMode := FALSE; END_IF;
   #"ioHMI-M".xButtonGoTo := #ixExtFullOpen AND "Clock_0.5Hz";
   #_w1 := #ixExtFullOpen AND NOT #sxForF5;   // rising edge of #ixExtFullOpen
   #sxForF5 := #ixExtFullOpen;
   IF #_w1 THEN #"ioHMI-M".xSwitchAutoMode := TRUE; END_IF;
END_REGION

REGION Network 26: Режим управления механизмом
   // 10 - местный
   // 20 - дистанционный ручной
   // 30 - дистанционный автоматический
   RUNG wire#powerrail
      I_Contact( #ixRemoteContr )
      Move(in := 10, out1 => #"ioHMI-M".wMode)
   END_RUNG
   RUNG wire#powerrail
      Contact( #ixRemoteContr )
      wire#w1
      I_Contact( #"ioHMI-M".xSwitchAutoMode )
      Move(in := 20, out1 => #"ioHMI-M".wMode)
   END_RUNG
   RUNG wire#w1
      Contact( #"ioHMI-M".xSwitchAutoMode )
      Move(in := 30, out1 => #"ioHMI-M".wMode)
   END_RUNG
   // the same network as SCL:
   IF NOT #ixRemoteContr THEN #"ioHMI-M".wMode := 10; END_IF;
   IF #ixRemoteContr AND NOT #"ioHMI-M".xSwitchAutoMode THEN #"ioHMI-M".wMode := 20; END_IF;
   IF #ixRemoteContr AND #"ioHMI-M".xSwitchAutoMode THEN #"ioHMI-M".wMode := 30; END_IF;
END_REGION

REGION Network 27: Код положения механизма
   // 10 - полностью открыт
   // 20 - промежуточное
   // 30 - полностью закрыт
   // 40 - оба концевика
   RUNG wire#powerrail
      Contact( #ixFullOpen )
      Move(in := 10, out1 => #"ioHMI-M".wPositionCode)
   END_RUNG
   RUNG wire#powerrail
      I_Contact( #ixFullOpen )
      I_Contact( #ixFullClose )
      Move(in := 20, out1 => #"ioHMI-M".wPositionCode)
   END_RUNG
   RUNG wire#powerrail
      Contact( #ixFullClose )
      Move(in := 30, out1 => #"ioHMI-M".wPositionCode)
   END_RUNG
   RUNG wire#powerrail
      Contact( #ixFullOpen )
      Contact( #ixFullClose )
      Move(in := 40, out1 => #"ioHMI-M".wPositionCode)
   END_RUNG
   // the same network as SCL:
   IF #ixFullOpen THEN #"ioHMI-M".wPositionCode := 10; END_IF;
   IF NOT #ixFullOpen AND NOT #ixFullClose THEN #"ioHMI-M".wPositionCode := 20; END_IF;
   IF #ixFullClose THEN #"ioHMI-M".wPositionCode := 30; END_IF;
   IF #ixFullOpen AND #ixFullClose THEN #"ioHMI-M".wPositionCode := 40; END_IF;
END_REGION

REGION Network 28: Код управления механизмом
   // 10 - нет команды на ход механизма
   // 20 - команда открыть
   // 30 - команда закрыть
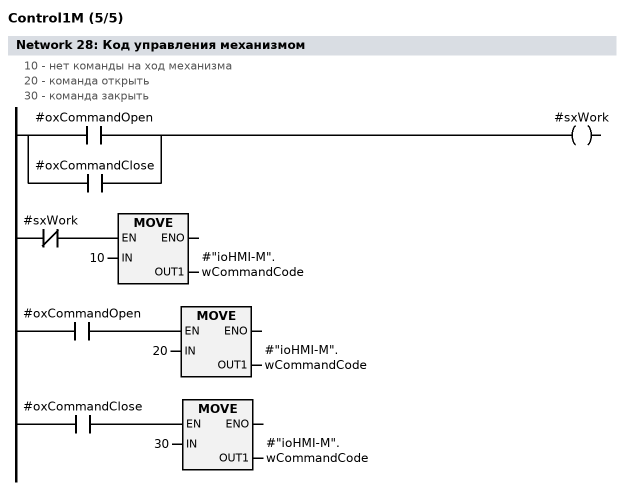
   RUNG wire#powerrail
      Contact( #oxCommandOpen )
      wire#w1
      Coil( #sxWork )
   END_RUNG
   RUNG wire#powerrail
      Contact( #oxCommandClose )
   END_RUNG wire#w1
   RUNG wire#powerrail
      I_Contact( #sxWork )
      Move(in := 10, out1 => #"ioHMI-M".wCommandCode)
   END_RUNG
   RUNG wire#powerrail
      Contact( #oxCommandOpen )
      Move(in := 20, out1 => #"ioHMI-M".wCommandCode)
   END_RUNG
   RUNG wire#powerrail
      Contact( #oxCommandClose )
      Move(in := 30, out1 => #"ioHMI-M".wCommandCode)
   END_RUNG
   // the same network as SCL:
   #sxWork := #oxCommandOpen OR #oxCommandClose;
   IF NOT #sxWork THEN #"ioHMI-M".wCommandCode := 10; END_IF;
   IF #oxCommandOpen THEN #"ioHMI-M".wCommandCode := 20; END_IF;
   IF #oxCommandClose THEN #"ioHMI-M".wCommandCode := 30; END_IF;
END_REGION
END_FUNCTION_BLOCK

FUNCTION_BLOCK "Control2M"   // FB502, LAD
TITLE = Управление Направляющим аппаратом 2М
{ S7_Optimized_Access := 'TRUE' }
VERSION : 0.1
   VAR_INPUT
      ixGuideReady : Bool;   // Готовность направляющего аппарата
      ixFullOpen : Bool;   // Полностью открыт
      ixFullClose : Bool;   // Полностью закрыт
      ixRemoteContr : Bool;   // Ключ в положении Дистанционный рехим
      ix2KM : Bool;   // Включен 2КМ1 или 2КМ2
      ixExtStop : Bool;   // Внешняя блокировка
      ixAutoModeCo : Bool;   // Авт.режим, 1=открыть, 0=закрыть
      ixAutoMoOpen : Bool;   // Авт.р., открыть (альтернатива ixAutoModeCo)
      ixAutoMoClose : Bool;   // Авт.р., закрыть (альтернатива ixAutoModeCo)
   END_VAR
   VAR_OUTPUT
      oxButOpen : Bool;   // Кнопка на ручное открытие
      oxButClose : Bool;   // Кнопка на ручное закрытие
      oxSwitchAutoMode : Bool;   // Переключатель (автомат.=1, ручной=0) на ЧМИ
      oxReady : Bool;   // Готовность механизма
      oxCommandOpen : Bool;   // Команда на открытие
      oxCommandClose : Bool;   // Команда на закрытие
   END_VAR
   VAR_IN_OUT
      "ioHMI-M" : "uHMI-Machine";   // Структура данных связи с ЧМИ
   END_VAR
   VAR
      sxWarning : Bool;   // Есть предупреждения
      sxFault : Bool;   // Есть авария
      sxWork : Bool;   // Есть моя команда
      sxForF1 : Bool;   // Статический бит для обнаружения фронта сигнала
      sxForF2 : Bool;   // Статический бит для обнаружения фронта сигнала
      sxForF3 : Bool;   // Статический бит для обнаружения фронта сигнала
      sxForF4 : Bool;   // Статический бит для обнаружения фронта сигнала
      sxForF5 : Bool;   // Статический бит для обнаружения фронта сигнала
      sxForF7 : Bool;   // Статический бит для обнаружения фронта сигнала
      sxForF8 : Bool;   // Статический бит для обнаружения фронта сигнала
      sxForF9 : Bool;   // Статический бит для обнаружения фронта сигнала
      sxForF10 : Bool;   // Статический бит для обнаружения фронта сигнала
      IEC_TimerInstance2 : TON_TIME;   // Таймер
      IEC_TimerInstance1 : TON_TIME;   // Таймер
      sxManOpen : Bool;   // Статический бит для команды открытия
      sxManClose : Bool;   // Статический бит для команды закрытия
      sxAutoOpen : Bool;   // Статический бит для команды открытия
      sxAutoClose : Bool;   // Статический бит для команды закрытия
      sxAutoOpen2 : Bool;   // Статический бит для команды открытия
      sxAutoClose2 : Bool;   // Статический бит для команды закрытия
   END_VAR
   VAR_TEMP
      tx1 : Bool;   // Временный бит
      tx2 : Bool;   // Временный бит
   END_VAR
   VAR_TEMP   // added for the SCL form of the ladder/FBD networks
      _w1 : Bool;
      _w2 : Bool;
      _w3 : Bool;
      _w4 : Bool;
      _w5 : Bool;
      _w6 : Bool;
      _w7 : Bool;
      _w8 : Bool;
   END_VAR
BEGIN

REGION Network 4: Подготовка данных от HMI:
END_REGION

REGION Network 5 (SCL): -виртуальные кнопки
   #oxButOpen  :=  #"ioHMI-M".xButManOpen;
   #oxButClose  :=  #"ioHMI-M".xButManClose;

   #oxSwitchAutoMode := #"ioHMI-M".xSwitchAutoMode;
END_REGION

REGION Network 7: ПРЕДУПРЕЖДЕНИЯ 2М (для журнала предупреждений на ЧМИ)
   // //wWarnings.%X0 - полностью закрыт
   // //wWarnings.%X1 - полностью открыт
   // wWarnings.%X2 - нет готовности от механизма  (было в дистанционном режиме, с 27.12.2020 - во всех режимах)
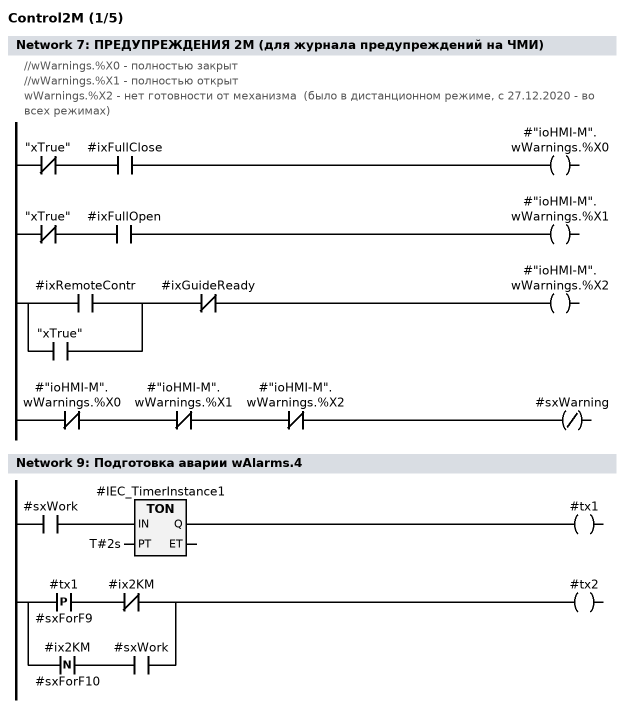
   RUNG wire#powerrail
      I_Contact( "xTrue" )
      Contact( #ixFullClose )
      Coil( #"ioHMI-M".wWarnings.%X0 )
   END_RUNG
   RUNG wire#powerrail
      I_Contact( "xTrue" )
      Contact( #ixFullOpen )
      Coil( #"ioHMI-M".wWarnings.%X1 )
   END_RUNG
   RUNG wire#powerrail
      Contact( #ixRemoteContr )
      wire#w1
      I_Contact( #ixGuideReady )
      Coil( #"ioHMI-M".wWarnings.%X2 )
   END_RUNG
   RUNG wire#powerrail
      Contact( "xTrue" )
   END_RUNG wire#w1
   RUNG wire#powerrail
      I_Contact( #"ioHMI-M".wWarnings.%X0 )
      I_Contact( #"ioHMI-M".wWarnings.%X1 )
      I_Contact( #"ioHMI-M".wWarnings.%X2 )
      I_Coil( #sxWarning )
   END_RUNG
   // the same network as SCL:
   #"ioHMI-M".wWarnings.%X0 := NOT "xTrue" AND #ixFullClose;
   #"ioHMI-M".wWarnings.%X1 := NOT "xTrue" AND #ixFullOpen;
   #"ioHMI-M".wWarnings.%X2 := (#ixRemoteContr OR "xTrue") AND NOT #ixGuideReady;
   #sxWarning := NOT (NOT #"ioHMI-M".wWarnings.%X0 AND NOT #"ioHMI-M".wWarnings.%X1 AND NOT #"ioHMI-M".wWarnings.%X2);
END_REGION

REGION Network 9: Подготовка аварии wAlarms.4
   #IEC_TimerInstance1(IN := #sxWork, PT := T#2s);   // TON
   #tx1 := #IEC_TimerInstance1.Q;
   #_w1 := #tx1 AND NOT #sxForF9;   // rising edge of #tx1
   #sxForF9 := #tx1;
   #_w2 := NOT #ix2KM AND #sxForF10;   // falling edge of #ix2KM
   #sxForF10 := #ix2KM;
   #tx2 := (#_w1 AND NOT #ix2KM) OR (#_w2 AND #sxWork);
END_REGION

REGION Network 10: АВАРИИ (для журнала аварийных сообщений на ЧМИ)
   // wAlarms.0 - одновременно оба концевика
   // wAlarms.1 - пропала готовность МЭО при работе
   // wAlarms.2 - команда не снимается более 1/2мин
   // wAlarms.3 - ход механизма без моей команды 
   // wAlarms.4 - моя команда есть, а пускателя нет
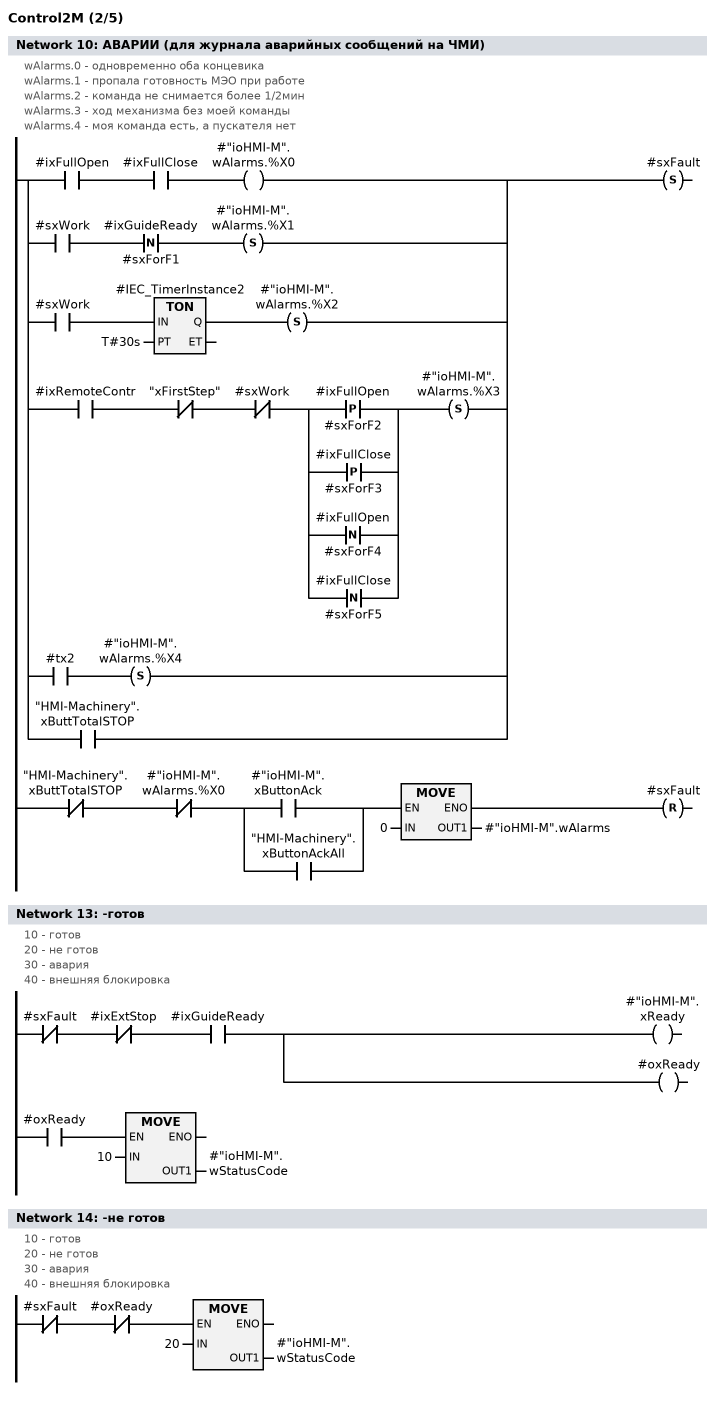
   #"ioHMI-M".wAlarms.%X0 := #ixFullOpen AND #ixFullClose;
   #_w1 := #sxWork AND NOT #ixGuideReady AND #sxForF1;   // falling edge of #ixGuideReady
   #sxForF1 := #ixGuideReady;
   #_w2 := #"ioHMI-M".wAlarms.%X0;
   IF #_w1 THEN #"ioHMI-M".wAlarms.%X1 := TRUE; END_IF;
   #IEC_TimerInstance2(IN := #sxWork, PT := T#30s);   // TON
   IF #IEC_TimerInstance2.Q THEN #"ioHMI-M".wAlarms.%X2 := TRUE; END_IF;
   #_w3 := #ixRemoteContr AND NOT "xFirstStep" AND NOT #sxWork AND #ixFullOpen AND NOT #sxForF2;   // rising edge of #ixFullOpen
   #sxForF2 := #ixFullOpen;
   #_w4 := #ixRemoteContr AND NOT "xFirstStep" AND NOT #sxWork AND #ixFullClose AND NOT #sxForF3;   // rising edge of #ixFullClose
   #sxForF3 := #ixFullClose;
   #_w5 := #ixRemoteContr AND NOT "xFirstStep" AND NOT #sxWork AND NOT #ixFullOpen AND #sxForF4;   // falling edge of #ixFullOpen
   #sxForF4 := #ixFullOpen;
   #_w6 := #ixRemoteContr AND NOT "xFirstStep" AND NOT #sxWork AND NOT #ixFullClose AND #sxForF5;   // falling edge of #ixFullClose
   #sxForF5 := #ixFullClose;
   #_w7 := #_w3 OR #_w4 OR #_w5 OR #_w6;
   IF #_w7 THEN #"ioHMI-M".wAlarms.%X3 := TRUE; END_IF;
   IF #tx2 THEN #"ioHMI-M".wAlarms.%X4 := TRUE; END_IF;
   IF #_w2 OR #_w1 OR #IEC_TimerInstance2.Q OR #_w7 OR #tx2 OR "HMI-Machinery".xButtTotalSTOP THEN
       #sxFault := TRUE;
   END_IF;
   #_w8 := NOT "HMI-Machinery".xButtTotalSTOP AND NOT #"ioHMI-M".wAlarms.%X0 AND (#"ioHMI-M".xButtonAck OR "HMI-Machinery".xButtonAckAll);
   IF #_w8 THEN
       #"ioHMI-M".wAlarms := 0;
       #sxFault := FALSE;
   END_IF;
END_REGION

REGION Network 12: Статус/состояние механизма:
END_REGION

REGION Network 13: -готов
   // 10 - готов
   // 20 - не готов
   // 30 - авария
   // 40 - внешняя блокировка
   RUNG wire#powerrail
      I_Contact( #sxFault )
      I_Contact( #ixExtStop )
      Contact( #ixGuideReady )
      wire#w1
      Coil( #"ioHMI-M".xReady )
   END_RUNG
   RUNG wire#w1
      Coil( #oxReady )
   END_RUNG
   RUNG wire#powerrail
      Contact( #oxReady )
      Move(in := 10, out1 => #"ioHMI-M".wStatusCode)
   END_RUNG
   // the same network as SCL:
   #"ioHMI-M".xReady := NOT #sxFault AND NOT #ixExtStop AND #ixGuideReady;
   #oxReady := #"ioHMI-M".xReady;
   IF #oxReady THEN #"ioHMI-M".wStatusCode := 10; END_IF;
END_REGION

REGION Network 14: -не готов
   // 10 - готов
   // 20 - не готов
   // 30 - авария
   // 40 - внешняя блокировка
   RUNG wire#powerrail
      I_Contact( #sxFault )
      I_Contact( #oxReady )
      Move(in := 20, out1 => #"ioHMI-M".wStatusCode)
   END_RUNG
   // the same network as SCL:
   IF NOT #sxFault AND NOT #oxReady THEN #"ioHMI-M".wStatusCode := 20; END_IF;
END_REGION

REGION Network 15: -авария
   // 10 - готов
   // 20 - не готов
   // 30 - авария
   // 40 - внешняя блокировка
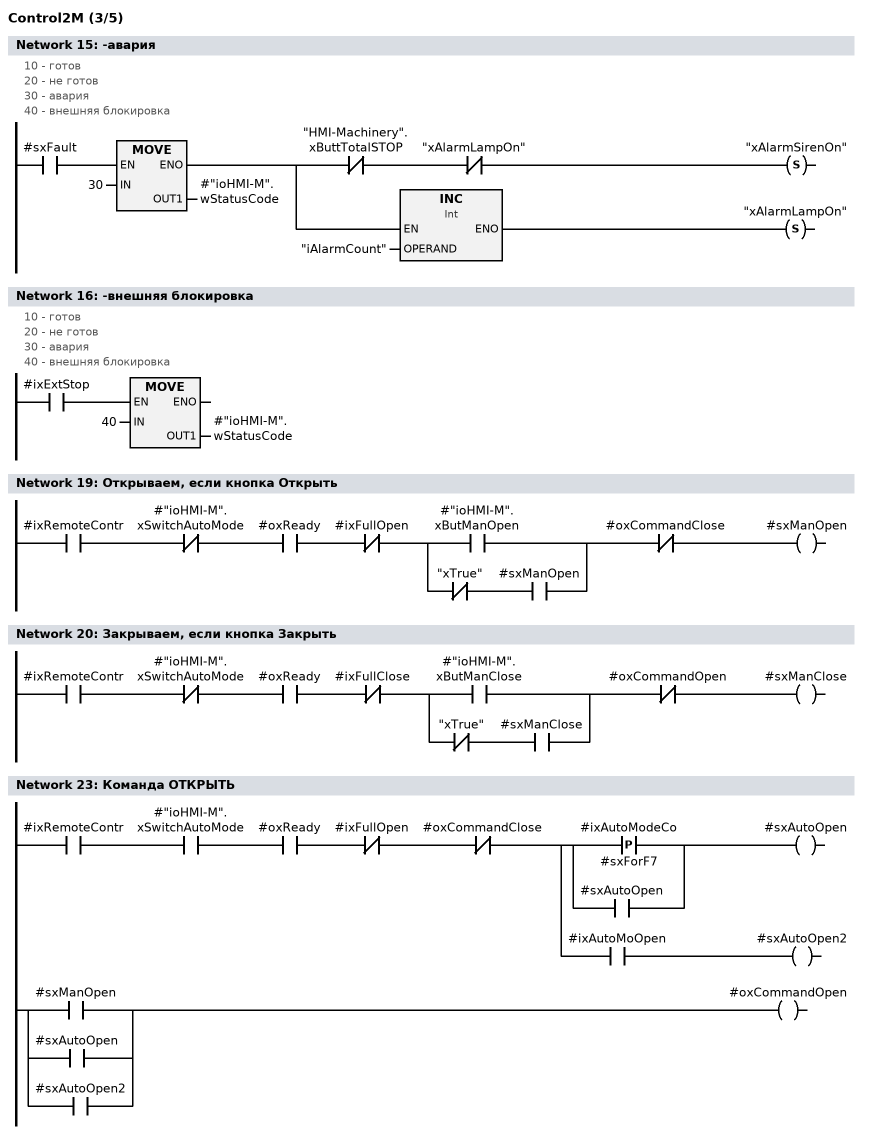
   RUNG wire#powerrail
      Contact( #sxFault )
      Move(in := 30, out1 => #"ioHMI-M".wStatusCode)
      wire#w1
      I_Contact( "HMI-Machinery".xButtTotalSTOP )
      I_Contact( "xAlarmLampOn" )
      S_Coil( "xAlarmSirenOn" )
   END_RUNG
   RUNG wire#w1
      { S7_Templates := "DestType := Int" } Inc( "iAlarmCount" )
      S_Coil( "xAlarmLampOn" )
   END_RUNG
   // the same network as SCL:
   IF #sxFault THEN #"ioHMI-M".wStatusCode := 30; END_IF;
   IF #sxFault AND NOT "HMI-Machinery".xButtTotalSTOP AND NOT "xAlarmLampOn" THEN
       "xAlarmSirenOn" := TRUE;
   END_IF;
   IF #sxFault THEN
       "iAlarmCount" := "iAlarmCount" + 1;
       "xAlarmLampOn" := TRUE;
   END_IF;
END_REGION

REGION Network 16: -внешняя блокировка
   // 10 - готов
   // 20 - не готов
   // 30 - авария
   // 40 - внешняя блокировка
   RUNG wire#powerrail
      Contact( #ixExtStop )
      Move(in := 40, out1 => #"ioHMI-M".wStatusCode)
   END_RUNG
   // the same network as SCL:
   IF #ixExtStop THEN #"ioHMI-M".wStatusCode := 40; END_IF;
END_REGION

REGION Network 18: Дистанционный РУЧНОЙ:
END_REGION

REGION Network 19: Открываем, если кнопка Открыть
   RUNG wire#powerrail
      Contact( #ixRemoteContr )
      I_Contact( #"ioHMI-M".xSwitchAutoMode )
      Contact( #oxReady )
      I_Contact( #ixFullOpen )
      wire#w1
      Contact( #"ioHMI-M".xButManOpen )
      wire#w2
      I_Contact( #oxCommandClose )
      Coil( #sxManOpen )
   END_RUNG
   RUNG wire#w1
      I_Contact( "xTrue" )
      Contact( #sxManOpen )
   END_RUNG wire#w2
   // the same network as SCL:
   #sxManOpen := #ixRemoteContr AND NOT #"ioHMI-M".xSwitchAutoMode AND #oxReady AND NOT #ixFullOpen AND (#"ioHMI-M".xButManOpen OR (NOT "xTrue" AND #sxManOpen)) AND NOT #oxCommandClose;
END_REGION

REGION Network 20: Закрываем, если кнопка Закрыть
   RUNG wire#powerrail
      Contact( #ixRemoteContr )
      I_Contact( #"ioHMI-M".xSwitchAutoMode )
      Contact( #oxReady )
      I_Contact( #ixFullClose )
      wire#w1
      Contact( #"ioHMI-M".xButManClose )
      wire#w2
      I_Contact( #oxCommandOpen )
      Coil( #sxManClose )
   END_RUNG
   RUNG wire#w1
      I_Contact( "xTrue" )
      Contact( #sxManClose )
   END_RUNG wire#w2
   // the same network as SCL:
   #sxManClose := #ixRemoteContr AND NOT #"ioHMI-M".xSwitchAutoMode AND #oxReady AND NOT #ixFullClose AND (#"ioHMI-M".xButManClose OR (NOT "xTrue" AND #sxManClose)) AND NOT #oxCommandOpen;
END_REGION

REGION Network 22: Дистанционный АВТОМАТИЧЕСКИЙ:
END_REGION

REGION Network 23: Команда ОТКРЫТЬ
   RUNG wire#powerrail
      Contact( #ixRemoteContr )
      Contact( #"ioHMI-M".xSwitchAutoMode )
      Contact( #oxReady )
      I_Contact( #ixFullOpen )
      I_Contact( #oxCommandClose )
      wire#w1
      P_Contact(operand := #ixAutoModeCo, bit := #sxForF7)
      wire#w2
      Coil( #sxAutoOpen )
   END_RUNG
   RUNG wire#w1
      Contact( #sxAutoOpen )
   END_RUNG wire#w2
   RUNG wire#w1
      Contact( #ixAutoMoOpen )
      Coil( #sxAutoOpen2 )
   END_RUNG
   RUNG wire#powerrail
      Contact( #sxManOpen )
      wire#w3
      Coil( #oxCommandOpen )
   END_RUNG
   RUNG wire#powerrail
      Contact( #sxAutoOpen )
   END_RUNG wire#w3
   RUNG wire#powerrail
      Contact( #sxAutoOpen2 )
   END_RUNG wire#w3
   // the same network as SCL:
   #_w1 := #ixRemoteContr AND #"ioHMI-M".xSwitchAutoMode AND #oxReady AND NOT #ixFullOpen AND NOT #oxCommandClose;
   #_w2 := #_w1 AND #ixAutoModeCo AND NOT #sxForF7;   // rising edge of #ixAutoModeCo
   #sxForF7 := #ixAutoModeCo;
   #sxAutoOpen := #_w2 OR (#_w1 AND #sxAutoOpen);
   #sxAutoOpen2 := #_w1 AND #ixAutoMoOpen;
   #oxCommandOpen := #sxManOpen OR #sxAutoOpen OR #sxAutoOpen2;
END_REGION

REGION Network 24: Команда ЗАКРЫТЬ
